LIN {X 0,Y 440.181,Z 736.749,A -85,B 0,C 180,E1 21310.496,E2 21310.496} C_VEL
LIN {X 0,Y 440.061,Z 740.552,A -85,B 0,C 180,E1 21308.405,E2 21308.405} C_VEL
LIN {X 0,Y 440.015,Z 742.533,A -85,B 0,C 180,E1 21306.286,E2 21306.286} C_VEL
LIN {X 0,Y 440.014,Z 742.803,A -85,B 0,C 180,E1 21304.135,E2 21304.135} C_VEL
LIN {X 0,Y 440.046,Z 741.335,A -85,B 0,C 180,E1 21302.093,E2 21302.093} C_VEL
LIN {X 0,Y 440.151,Z 738.009,A -85,B 0,C 180,E1 21299.94,E2 21299.94} C_VEL
LIN {X 0,Y 440.36,Z 733.034,A -85,B 0,C 180,E1 21297.908,E2 21297.908} C_VEL
LIN {X 0,Y 440.738,Z 726.189,A -85,B 0,C 180,E1 21295.899,E2 21295.899} C_VEL
LIN {X 0,Y 441.277,Z 718.01,A -85,B 0,C 180,E1 21294.069,E2 21294.069} C_VEL
LIN {X 0,Y 442.008,Z 707.793,A -85,B 0,C 180,E1 21292.276,E2 21292.276} C_VEL
LIN {X 0,Y 442.843,Z 696.61,A -85,B 0,C 180,E1 21290.715,E2 21290.715} C_VEL
LIN {X 0,Y 443.748,Z 683.902,A -85,B 0,C 180,E1 21289.299,E2 21289.299} C_VEL
LIN {X 0,Y 444.656,Z 670.333,A -85,B 0,C 180,E1 21288.099,E2 21288.099} C_VEL
LIN {X 0,Y 445.545,Z 654.948,A -85,B 0,C 180,E1 21287.053,E2 21287.053} C_VEL
LIN {X 0,Y 446.221,Z 639.636,A -85,B 0,C 180,E1 21286.284,E2 21286.284} C_VEL
LIN {X 0,Y 446.712,Z 622.753,A -85,B 0,C 180,E1 21285.709,E2 21285.709} C_VEL
LIN {X 0,Y 447.044,Z 598.324,A -85,B 0,C 180,E1 21285.256,E2 21285.256} C_VEL
LIN {X 0,Y 448.29,Z 488.008,A -85,B 0,C 180,E1 21283.44,E2 21283.44} C_VEL
LIN {X 0,Y 447.015,Z 476.916,A -85,B 0,C 180,E1 21283.152,E2 21283.152} C_VEL
LIN {X 0,Y 448.557,Z 433.644,A -85,B 0,C 180,E1 21279.442,E2 21279.442} C_VEL
LIN {X 0,Y 450.183,Z 391.513,A -85,B 0,C 180,E1 21275.842,E2 21275.842} C_VEL
LIN {X 0,Y 451.444,Z 352.894,A -85,B 0,C 180,E1 21272.562,E2 21272.562} C_VEL
LIN {X 0,Y 452.462,Z 314.159,A -85,B 0,C 180,E1 21269.27,E2 21269.27} C_VEL
LIN {X 0,Y 446.407,Z 295.705,A -85,B 0,C 180,E1 21267.189,E2 21267.189} C_VEL
LIN {X 0,Y 441.254,Z 281.906,A -85,B 0,C 180,E1 21265.502,E2 21265.502} C_VEL
LIN {X 0,Y 441.178,Z 281.529,A -85,B 0,C 180,E1 21265.076,E2 21265.076} C_VEL
LIN {X 0,Y 441.198,Z 281.522,A -85,B 0,C 180,E1 21261.348,E2 21261.348} C_VEL
LIN {X 0,Y 441.197,Z 281.527,A -85,B 0,C 180,E1 21257.543,E2 21257.543} C_VEL
LIN {X 0,Y 441.185,Z 281.533,A -85,B 0,C 180,E1 21253.767,E2 21253.767} C_VEL
LIN {X 0,Y 441.166,Z 281.531,A -85,B 0,C 180,E1 21250.051,E2 21250.051} C_VEL
LIN {X 0,Y 441.16,Z 281.529,A -85,B 0,C 180,E1 21246.377,E2 21246.377} C_VEL
LIN {X 0,Y 441.167,Z 281.529,A -85,B 0,C 180,E1 21242.598,E2 21242.598} C_VEL
LIN {X 0,Y 441.191,Z 281.524,A -85,B 0,C 180,E1 21238.962,E2 21238.962} C_VEL
LIN {X 0,Y 441.199,Z 281.529,A -85,B 0,C 180,E1 21235.191,E2 21235.191} C_VEL
LIN {X 0,Y 441.196,Z 281.528,A -85,B 0,C 180,E1 21231.398,E2 21231.398} C_VEL
LIN {X 0,Y 441.18,Z 281.528,A -85,B 0,C 180,E1 21227.621,E2 21227.621} C_VEL
LIN {X 0,Y 441.166,Z 281.526,A -85,B 0,C 180,E1 21223.928,E2 21223.928} C_VEL
LIN {X 0,Y 441.164,Z 281.528,A -85,B 0,C 180,E1 21220.126,E2 21220.126} C_VEL
LIN {X 0,Y 441.173,Z 281.528,A -85,B 0,C 180,E1 21216.351,E2 21216.351} C_VEL
LIN {X 0,Y 441.191,Z 281.525,A -85,B 0,C 180,E1 21212.61,E2 21212.61} C_VEL
LIN {X 0,Y 441.201,Z 281.527,A -85,B 0,C 180,E1 21208.889,E2 21208.889} C_VEL
LIN {X 0,Y 441.198,Z 281.531,A -85,B 0,C 180,E1 21205.119,E2 21205.119} C_VEL
LIN {X 0,Y 441.192,Z 281.531,A -85,B 0,C 180,E1 21201.282,E2 21201.282} C_VEL
LIN {X 0,Y 441.177,Z 281.532,A -85,B 0,C 180,E1 21197.518,E2 21197.518} C_VEL
LIN {X 0,Y 441.171,Z 281.531,A -85,B 0,C 180,E1 21193.726,E2 21193.726} C_VEL
LIN {X 0,Y 441.247,Z 281.87,A -85,B 0,C 180,E1 21192.618,E2 21192.618} C_VEL
LIN {X 0,Y 450.274,Z 303.715,A -85,B 0,C 180,E1 21189.499,E2 21189.499} C_VEL
LIN {X 0,Y 455.991,Z 317.99,A -85,B 0,C 180,E1 21187.668,E2 21187.668} C_VEL
LIN {X 0,Y 460.666,Z 327.189,A -85,B 0,C 180,E1 21187.056,E2 21187.056} C_VEL
LIN {X 0,Y 462.807,Z 343.497,A -85,B 0,C 180,E1 21186.538,E2 21186.538} C_VEL
LIN {X 0,Y 457.811,Z 535.941,A -85,B 0,C 180,E1 21183.072,E2 21183.072} C_VEL
LIN {X 0,Y 456.712,Z 578.69,A -85,B 0,C 180,E1 21182.281,E2 21182.281} C_VEL
LIN {X 0,Y 455.661,Z 599.497,A -85,B 0,C 180,E1 21181.679,E2 21181.679} C_VEL
LIN {X 0,Y 454.252,Z 620.653,A -85,B 0,C 180,E1 21180.816,E2 21180.816} C_VEL
LIN {X 0,Y 452.631,Z 640.786,A -85,B 0,C 180,E1 21179.736,E2 21179.736} C_VEL
LIN {X 0,Y 450.918,Z 659.614,A -85,B 0,C 180,E1 21178.471,E2 21178.471} C_VEL
LIN {X 0,Y 449.126,Z 677.545,A -85,B 0,C 180,E1 21177.008,E2 21177.008} C_VEL
LIN {X 0,Y 447.343,Z 694.663,A -85,B 0,C 180,E1 21175.334,E2 21175.334} C_VEL
LIN {X 0,Y 445.58,Z 711.241,A -85,B 0,C 180,E1 21173.398,E2 21173.398} C_VEL
LIN {X 0,Y 444.067,Z 725.727,A -85,B 0,C 180,E1 21171.391,E2 21171.391} C_VEL
LIN {X 0,Y 442.781,Z 738.828,A -85,B 0,C 180,E1 21169.248,E2 21169.248} C_VEL
LIN {X 0,Y 441.743,Z 750.531,A -85,B 0,C 180,E1 21166.975,E2 21166.975} C_VEL
LIN {X 0,Y 440.958,Z 760.738,A -85,B 0,C 180,E1 21164.576,E2 21164.576} C_VEL
LIN {X 0,Y 440.444,Z 769.059,A -85,B 0,C 180,E1 21162.186,E2 21162.186} C_VEL
LIN {X 0,Y 440.125,Z 776.357,A -85,B 0,C 180,E1 21159.544,E2 21159.544} C_VEL
LIN {X 0,Y 439.984,Z 781.551,A -85,B 0,C 180,E1 21157.047,E2 21157.047} C_VEL
LIN {X 0,Y 439.941,Z 785.113,A -85,B 0,C 180,E1 21154.561,E2 21154.561} C_VEL
LIN {X 0,Y 439.94,Z 787.077,A -85,B 0,C 180,E1 21152.082,E2 21152.082} C_VEL
LIN {X 0,Y 439.937,Z 787.552,A -85,B 0,C 180,E1 21149.478,E2 21149.478} C_VEL
LIN {X 0,Y 439.937,Z 786.489,A -85,B 0,C 180,E1 21147.002,E2 21147.002} C_VEL
LIN {X 0,Y 439.952,Z 783.805,A -85,B 0,C 180,E1 21144.513,E2 21144.513} C_VEL
LIN {X 0,Y 440.044,Z 779.312,A -85,B 0,C 180,E1 21141.9,E2 21141.9} C_VEL
LIN {X 0,Y 440.252,Z 772.933,A -85,B 0,C 180,E1 21139.266,E2 21139.266} C_VEL
LIN {X 0,Y 440.634,Z 764.984,A -85,B 0,C 180,E1 21136.75,E2 21136.75} C_VEL
LIN {X 0,Y 441.243,Z 755.554,A -85,B 0,C 180,E1 21134.355,E2 21134.355} C_VEL
LIN {X 0,Y 442.122,Z 743.965,A -85,B 0,C 180,E1 21131.95,E2 21131.95} C_VEL
LIN {X 0,Y 443.172,Z 731.504,A -85,B 0,C 180,E1 21129.805,E2 21129.805} C_VEL
LIN {X 0,Y 444.435,Z 717.672,A -85,B 0,C 180,E1 21127.792,E2 21127.792} C_VEL
LIN {X 0,Y 445.876,Z 702.126,A -85,B 0,C 180,E1 21125.878,E2 21125.878} C_VEL
LIN {X 0,Y 447.474,Z 684.889,A -85,B 0,C 180,E1 21124.097,E2 21124.097} C_VEL
LIN {X 0,Y 449.047,Z 666.984,A -85,B 0,C 180,E1 21122.553,E2 21122.553} C_VEL
LIN {X 0,Y 450.605,Z 648.2,A -85,B 0,C 180,E1 21121.215,E2 21121.215} C_VEL
LIN {X 0,Y 452.045,Z 628.603,A -85,B 0,C 180,E1 21120.08,E2 21120.08} C_VEL
LIN {X 0,Y 453.369,Z 607.681,A -85,B 0,C 180,E1 21119.133,E2 21119.133} C_VEL
LIN {X 0,Y 454.47,Z 585.842,A -85,B 0,C 180,E1 21118.407,E2 21118.407} C_VEL
LIN {X 0,Y 455.219,Z 563.267,A -85,B 0,C 180,E1 21117.912,E2 21117.912} C_VEL
LIN {X 0,Y 457.443,Z 471.715,A -85,B 0,C 180,E1 21116.219,E2 21116.219} C_VEL
LIN {X 0,Y 460.734,Z 385.677,A -85,B 0,C 180,E1 21114.431,E2 21114.431} C_VEL
LIN {X 0,Y 462.815,Z 341.137,A -85,B 0,C 180,E1 21113.409,E2 21113.409} C_VEL
LIN {X 0,Y 461.409,Z 327.079,A -85,B 0,C 180,E1 21112.807,E2 21112.807} C_VEL
LIN {X 0,Y 459.208,Z 322.242,A -85,B 0,C 180,E1 21112.322,E2 21112.322} C_VEL
LIN {X 0,Y 456.915,Z 314.351,A -85,B 0,C 180,E1 21110.932,E2 21110.932} C_VEL
LIN {X 0,Y 454.658,Z 308.19,A -85,B 0,C 180,E1 21109.543,E2 21109.543} C_VEL
LIN {X 0,Y 453.091,Z 304.346,A -85,B 0,C 180,E1 21108.425,E2 21108.425} C_VEL
LIN {X 0,Y 451.999,Z 301.525,A -85,B 0,C 180,E1 21107.397,E2 21107.397} C_VEL
LIN {X 0,Y 450.664,Z 298.499,A -85,B 0,C 180,E1 21105.594,E2 21105.594} C_VEL
LIN {X 0,Y 450.382,Z 297.678,A -85,B 0,C 180,E1 21104.549,E2 21104.549} C_VEL
LIN {X 0,Y 450.505,Z 297.961,A -85,B 0,C 180,E1 21102.91,E2 21102.91} C_VEL
LIN {X 0,Y 451.405,Z 300.859,A -85,B 0,C 180,E1 21100.946,E2 21100.946} C_VEL
LIN {X 0,Y 452.242,Z 302.678,A -85,B 0,C 180,E1 21100.095,E2 21100.095} C_VEL
LIN {X 0,Y 453.759,Z 306.663,A -85,B 0,C 180,E1 21098.735,E2 21098.735} C_VEL
LIN {X 0,Y 455.605,Z 311.582,A -85,B 0,C 180,E1 21097.397,E2 21097.397} C_VEL
LIN {X 0,Y 458.153,Z 319.894,A -85,B 0,C 180,E1 21095.64,E2 21095.64} C_VEL
LIN {X 0,Y 459.651,Z 326.416,A -85,B 0,C 180,E1 21094.509,E2 21094.509} C_VEL
LIN {X 0,Y 458.028,Z 338.193,A -85,B 0,C 180,E1 21093.261,E2 21093.261} C_VEL
LIN {X 0,Y 460.688,Z 358.394,A -85,B 0,C 180,E1 21092.208,E2 21092.208} C_VEL
LIN {X 0,Y 461.626,Z 369.193,A -85,B 0,C 180,E1 21091.757,E2 21091.757} C_VEL
LIN {X 0,Y 456.809,Z 456.691,A -85,B 0,C 180,E1 21089.751,E2 21089.751} C_VEL
LIN {X 0,Y 453.689,Z 542.646,A -85,B 0,C 180,E1 21087.956,E2 21087.956} C_VEL
LIN {X 0,Y 452.772,Z 568.529,A -85,B 0,C 180,E1 21087.378,E2 21087.378} C_VEL
LIN {X 0,Y 451.765,Z 588.323,A -85,B 0,C 180,E1 21086.697,E2 21086.697} C_VEL
LIN {X 0,Y 450.577,Z 606.905,A -85,B 0,C 180,E1 21085.828,E2 21085.828} C_VEL
LIN {X 0,Y 449.224,Z 625.06,A -85,B 0,C 180,E1 21084.736,E2 21084.736} C_VEL
LIN {X 0,Y 447.734,Z 642.969,A -85,B 0,C 180,E1 21083.388,E2 21083.388} C_VEL
LIN {X 0,Y 446.223,Z 659.644,A -85,B 0,C 180,E1 21081.836,E2 21081.836} C_VEL
LIN {X 0,Y 444.779,Z 674.825,A -85,B 0,C 180,E1 21080.117,E2 21080.117} C_VEL
LIN {X 0,Y 443.489,Z 688.388,A -85,B 0,C 180,E1 21078.263,E2 21078.263} C_VEL
LIN {X 0,Y 442.379,Z 700.441,A -85,B 0,C 180,E1 21076.275,E2 21076.275} C_VEL
LIN {X 0,Y 441.483,Z 711.005,A -85,B 0,C 180,E1 21074.158,E2 21074.158} C_VEL
LIN {X 0,Y 440.847,Z 719.619,A -85,B 0,C 180,E1 21072.043,E2 21072.043} C_VEL
LIN {X 0,Y 440.381,Z 727.255,A -85,B 0,C 180,E1 21069.672,E2 21069.672} C_VEL
LIN {X 0,Y 440.121,Z 733.018,A -85,B 0,C 180,E1 21067.309,E2 21067.309} C_VEL
LIN {X 0,Y 439.997,Z 737.235,A -85,B 0,C 180,E1 21064.823,E2 21064.823} C_VEL
LIN {X 0,Y 439.954,Z 739.675,A -85,B 0,C 180,E1 21062.344,E2 21062.344} C_VEL
LIN {X 0,Y 439.951,Z 740.425,A -85,B 0,C 180,E1 21059.869,E2 21059.869} C_VEL
LIN {X 0,Y 439.953,Z 739.489,A -85,B 0,C 180,E1 21057.394,E2 21057.394} C_VEL
LIN {X 0,Y 439.993,Z 736.836,A -85,B 0,C 180,E1 21054.915,E2 21054.915} C_VEL
LIN {X 0,Y 440.118,Z 732.414,A -85,B 0,C 180,E1 21052.428,E2 21052.428} C_VEL
LIN {X 0,Y 440.407,Z 726.08,A -85,B 0,C 180,E1 21049.932,E2 21049.932} C_VEL
LIN {X 0,Y 440.892,Z 718.138,A -85,B 0,C 180,E1 21047.558,E2 21047.558} C_VEL
LIN {X 0,Y 441.611,Z 708.667,A -85,B 0,C 180,E1 21045.31,E2 21045.31} C_VEL
LIN {X 0,Y 442.571,Z 697.708,A -85,B 0,C 180,E1 21043.191,E2 21043.191} C_VEL
LIN {X 0,Y 443.755,Z 685.267,A -85,B 0,C 180,E1 21041.203,E2 21041.203} C_VEL
LIN {X 0,Y 445.136,Z 671.283,A -85,B 0,C 180,E1 21039.35,E2 21039.35} C_VEL
LIN {X 0,Y 446.614,Z 656.284,A -85,B 0,C 180,E1 21037.699,E2 21037.699} C_VEL
LIN {X 0,Y 448.114,Z 640.389,A -85,B 0,C 180,E1 21036.25,E2 21036.25} C_VEL
LIN {X 0,Y 449.573,Z 623.714,A -85,B 0,C 180,E1 21035.003,E2 21035.003} C_VEL
LIN {X 0,Y 450.969,Z 605.565,A -85,B 0,C 180,E1 21033.917,E2 21033.917} C_VEL
LIN {X 0,Y 452.193,Z 586.81,A -85,B 0,C 180,E1 21033.054,E2 21033.054} C_VEL
LIN {X 0,Y 453.148,Z 567.759,A -85,B 0,C 180,E1 21032.418,E2 21032.418} C_VEL
LIN {X 0,Y 453.837,Z 546.607,A -85,B 0,C 180,E1 21031.963,E2 21031.963} C_VEL
LIN {X 0,Y 458.256,Z 366.504,A -85,B 0,C 180,E1 21028.685,E2 21028.685} C_VEL
LIN {X 0,Y 454.172,Z 340.574,A -85,B 0,C 180,E1 21027.787,E2 21027.787} C_VEL
LIN {X 0,Y 455.736,Z 321.368,A -85,B 0,C 180,E1 21025.928,E2 21025.928} C_VEL
LIN {X 0,Y 449.365,Z 303.02,A -85,B 0,C 180,E1 21023.393,E2 21023.393} C_VEL
LIN {X 0,Y 442.233,Z 284.592,A -85,B 0,C 180,E1 21020.647,E2 21020.647} C_VEL
LIN {X 0,Y 441.199,Z 281.714,A -85,B 0,C 180,E1 21020.149,E2 21020.149} C_VEL
LIN {X 0,Y 441.193,Z 281.525,A -85,B 0,C 180,E1 21016.487,E2 21016.487} C_VEL
LIN {X 0,Y 441.195,Z 281.525,A -85,B 0,C 180,E1 21012.658,E2 21012.658} C_VEL
LIN {X 0,Y 441.192,Z 281.529,A -85,B 0,C 180,E1 21009.612,E2 21009.612} C_VEL
LIN {X 0,Y 440.226,Z 281.651,A -85,B 0,C 180,E1 21008.611,E2 21008.611} C_VEL
LIN {X 0,Y 433.688,Z 282.466,A -85,B 0,C 180,E1 21005.722,E2 21005.722} C_VEL
LIN {X 0,Y 433.246,Z 282.517,A -85,B 0,C 180,E1 21005.059,E2 21005.059} C_VEL
LIN {X 0,Y 433.246,Z 282.516,A -85,B 0,C 180,E1 21001.284,E2 21001.284} C_VEL
LIN {X 0,Y 433.248,Z 282.519,A -85,B 0,C 180,E1 20997.489,E2 20997.489} C_VEL
LIN {X 0,Y 433.251,Z 282.513,A -85,B 0,C 180,E1 20993.677,E2 20993.677} C_VEL
LIN {X 0,Y 433.259,Z 282.516,A -85,B 0,C 180,E1 20989.973,E2 20989.973} C_VEL
LIN {X 0,Y 433.254,Z 282.505,A -85,B 0,C 180,E1 20986.079,E2 20986.079} C_VEL
LIN {X 0,Y 433.248,Z 282.789,A -85,B 0,C 180,E1 20985.34,E2 20985.34} C_VEL
LIN {X 0,Y 440.653,Z 303.028,A -85,B 0,C 180,E1 20982.783,E2 20982.783} C_VEL
LIN {X 0,Y 445.747,Z 318.928,A -85,B 0,C 180,E1 20980.927,E2 20980.927} C_VEL
LIN {X 0,Y 444.169,Z 360.129,A -85,B 0,C 180,E1 20977.308,E2 20977.308} C_VEL
LIN {X 0,Y 442.449,Z 402.117,A -85,B 0,C 180,E1 20973.629,E2 20973.629} C_VEL
LIN {X 0,Y 440.609,Z 445.061,A -85,B 0,C 180,E1 20969.871,E2 20969.871} C_VEL
LIN {X 0,Y 439.376,Z 477.348,A -85,B 0,C 180,E1 20967.073,E2 20967.073} C_VEL
LIN {X 0,Y 440.893,Z 492.134,A -85,B 0,C 180,E1 20966.733,E2 20966.733} C_VEL
LIN {X 0,Y 439.134,Z 620.462,A -85,B 0,C 180,E1 20964.571,E2 20964.571} C_VEL
LIN {X 0,Y 438.677,Z 636.459,A -85,B 0,C 180,E1 20964.061,E2 20964.061} C_VEL
LIN {X 0,Y 437.958,Z 652.869,A -85,B 0,C 180,E1 20963.274,E2 20963.274} C_VEL
LIN {X 0,Y 437.106,Z 667.453,A -85,B 0,C 180,E1 20962.311,E2 20962.311} C_VEL
LIN {X 0,Y 436.156,Z 681.295,A -85,B 0,C 180,E1 20961.133,E2 20961.133} C_VEL
LIN {X 0,Y 435.218,Z 693.946,A -85,B 0,C 180,E1 20959.772,E2 20959.772} C_VEL
LIN {X 0,Y 434.264,Z 706.231,A -85,B 0,C 180,E1 20958.109,E2 20958.109} C_VEL
LIN {X 0,Y 433.495,Z 716.267,A -85,B 0,C 180,E1 20956.395,E2 20956.395} C_VEL
LIN {X 0,Y 432.856,Z 725.39,A -85,B 0,C 180,E1 20954.417,E2 20954.417} C_VEL
LIN {X 0,Y 432.451,Z 732.108,A -85,B 0,C 180,E1 20952.51,E2 20952.51} C_VEL
LIN {X 0,Y 432.186,Z 737.739,A -85,B 0,C 180,E1 20950.323,E2 20950.323} C_VEL
LIN {X 0,Y 432.068,Z 741.172,A -85,B 0,C 180,E1 20948.27,E2 20948.27} C_VEL
LIN {X 0,Y 432.025,Z 743.034,A -85,B 0,C 180,E1 20946.09,E2 20946.09} C_VEL
LIN {X 0,Y 432.025,Z 743.18,A -85,B 0,C 180,E1 20944.063,E2 20944.063} C_VEL
LIN {X 0,Y 432.067,Z 741.49,A -85,B 0,C 180,E1 20941.832,E2 20941.832} C_VEL
LIN {X 0,Y 432.191,Z 738.024,A -85,B 0,C 180,E1 20939.648,E2 20939.648} C_VEL
LIN {X 0,Y 432.442,Z 732.785,A -85,B 0,C 180,E1 20937.558,E2 20937.558} C_VEL
LIN {X 0,Y 432.872,Z 725.848,A -85,B 0,C 180,E1 20935.537,E2 20935.537} C_VEL
LIN {X 0,Y 433.495,Z 717.09,A -85,B 0,C 180,E1 20933.608,E2 20933.608} C_VEL
LIN {X 0,Y 434.261,Z 707.32,A -85,B 0,C 180,E1 20931.901,E2 20931.901} C_VEL
LIN {X 0,Y 435.168,Z 695.801,A -85,B 0,C 180,E1 20930.304,E2 20930.304} C_VEL
LIN {X 0,Y 436.161,Z 682.809,A -85,B 0,C 180,E1 20928.861,E2 20928.861} C_VEL
LIN {X 0,Y 437.14,Z 668.595,A -85,B 0,C 180,E1 20927.629,E2 20927.629} C_VEL
LIN {X 0,Y 438.03,Z 653.898,A -85,B 0,C 180,E1 20926.643,E2 20926.643} C_VEL
LIN {X 0,Y 438.742,Z 637.746,A -85,B 0,C 180,E1 20925.855,E2 20925.855} C_VEL
LIN {X 0,Y 439.21,Z 621.585,A -85,B 0,C 180,E1 20925.324,E2 20925.324} C_VEL
LIN {X 0,Y 439.971,Z 565.077,A -85,B 0,C 180,E1 20924.345,E2 20924.345} C_VEL
LIN {X 0,Y 440.868,Z 488.855,A -85,B 0,C 180,E1 20923.064,E2 20923.064} C_VEL
LIN {X 0,Y 439.554,Z 477.444,A -85,B 0,C 180,E1 20922.766,E2 20922.766} C_VEL
LIN {X 0,Y 441.159,Z 434.521,A -85,B 0,C 180,E1 20919.056,E2 20919.056} C_VEL
LIN {X 0,Y 443.037,Z 389.151,A -85,B 0,C 180,E1 20915.135,E2 20915.135} C_VEL
LIN {X 0,Y 444.504,Z 345.174,A -85,B 0,C 180,E1 20911.382,E2 20911.382} C_VEL
LIN {X 0,Y 445.246,Z 316.819,A -85,B 0,C 180,E1 20908.943,E2 20908.943} C_VEL
LIN {X 0,Y 438.945,Z 297.654,A -85,B 0,C 180,E1 20906.737,E2 20906.737} C_VEL
LIN {X 0,Y 433.278,Z 282.866,A -85,B 0,C 180,E1 20904.875,E2 20904.875} C_VEL
LIN {X 0,Y 433.223,Z 282.522,A -85,B 0,C 180,E1 20904.257,E2 20904.257} C_VEL
LIN {X 0,Y 433.219,Z 282.519,A -85,B 0,C 180,E1 20900.446,E2 20900.446} C_VEL
LIN {X 0,Y 433.221,Z 282.523,A -85,B 0,C 180,E1 20896.63,E2 20896.63} C_VEL
LIN {X 0,Y 433.239,Z 282.518,A -85,B 0,C 180,E1 20892.937,E2 20892.937} C_VEL
LIN {X 0,Y 433.257,Z 282.516,A -85,B 0,C 180,E1 20889.163,E2 20889.163} C_VEL
LIN {X 0,Y 433.258,Z 282.52,A -85,B 0,C 180,E1 20885.43,E2 20885.43} C_VEL
LIN {X 0,Y 433.25,Z 282.516,A -85,B 0,C 180,E1 20881.587,E2 20881.587} C_VEL
LIN {X 0,Y 433.231,Z 282.518,A -85,B 0,C 180,E1 20877.884,E2 20877.884} C_VEL
LIN {X 0,Y 433.223,Z 282.52,A -85,B 0,C 180,E1 20874.092,E2 20874.092} C_VEL
LIN {X 0,Y 433.225,Z 282.514,A -85,B 0,C 180,E1 20870.215,E2 20870.215} C_VEL
LIN {X 0,Y 433.229,Z 282.517,A -85,B 0,C 180,E1 20866.385,E2 20866.385} C_VEL
LIN {X 0,Y 433.247,Z 282.516,A -85,B 0,C 180,E1 20862.68,E2 20862.68} C_VEL
LIN {X 0,Y 433.262,Z 282.513,A -85,B 0,C 180,E1 20858.9,E2 20858.9} C_VEL
LIN {X 0,Y 433.261,Z 282.515,A -85,B 0,C 180,E1 20855.082,E2 20855.082} C_VEL
LIN {X 0,Y 433.263,Z 282.518,A -85,B 0,C 180,E1 20851.271,E2 20851.271} C_VEL
LIN {X 0,Y 433.242,Z 282.518,A -85,B 0,C 180,E1 20847.471,E2 20847.471} C_VEL
LIN {X 0,Y 433.229,Z 282.518,A -85,B 0,C 180,E1 20843.785,E2 20843.785} C_VEL
LIN {X 0,Y 433.231,Z 282.518,A -85,B 0,C 180,E1 20839.917,E2 20839.917} C_VEL
LIN {X 0,Y 433.24,Z 282.521,A -85,B 0,C 180,E1 20836.183,E2 20836.183} C_VEL
LIN {X 0,Y 433.28,Z 282.785,A -85,B 0,C 180,E1 20833.395,E2 20833.395} C_VEL
LIN {X 0,Y 442.336,Z 304.575,A -85,B 0,C 180,E1 20830.181,E2 20830.181} C_VEL
LIN {X 0,Y 447.798,Z 318.027,A -85,B 0,C 180,E1 20828.398,E2 20828.398} C_VEL
LIN {X 0,Y 454.373,Z 330.66,A -85,B 0,C 180,E1 20827.533,E2 20827.533} C_VEL
LIN {X 0,Y 456.144,Z 344.815,A -85,B 0,C 180,E1 20827.076,E2 20827.076} C_VEL
LIN {X 0,Y 450.988,Z 527.844,A -85,B 0,C 180,E1 20823.703,E2 20823.703} C_VEL
LIN {X 0,Y 449.614,Z 578.4,A -85,B 0,C 180,E1 20822.755,E2 20822.755} C_VEL
LIN {X 0,Y 448.508,Z 599.317,A -85,B 0,C 180,E1 20822.141,E2 20822.141} C_VEL
LIN {X 0,Y 447.058,Z 619.962,A -85,B 0,C 180,E1 20821.29,E2 20821.29} C_VEL
LIN {X 0,Y 445.444,Z 639.254,A -85,B 0,C 180,E1 20820.25,E2 20820.25} C_VEL
LIN {X 0,Y 443.639,Z 658.179,A -85,B 0,C 180,E1 20818.982,E2 20818.982} C_VEL
LIN {X 0,Y 441.751,Z 676.334,A -85,B 0,C 180,E1 20817.497,E2 20817.497} C_VEL
LIN {X 0,Y 439.792,Z 694.198,A -85,B 0,C 180,E1 20815.735,E2 20815.735} C_VEL
LIN {X 0,Y 437.917,Z 710.869,A -85,B 0,C 180,E1 20813.763,E2 20813.763} C_VEL
LIN {X 0,Y 436.365,Z 724.971,A -85,B 0,C 180,E1 20811.788,E2 20811.788} C_VEL
LIN {X 0,Y 434.99,Z 738.152,A -85,B 0,C 180,E1 20809.607,E2 20809.607} C_VEL
LIN {X 0,Y 433.82,Z 750.534,A -85,B 0,C 180,E1 20807.156,E2 20807.156} C_VEL
LIN {X 0,Y 432.96,Z 761.231,A -85,B 0,C 180,E1 20804.578,E2 20804.578} C_VEL
LIN {X 0,Y 432.416,Z 769.799,A -85,B 0,C 180,E1 20802.01,E2 20802.01} C_VEL
LIN {X 0,Y 432.115,Z 776.509,A -85,B 0,C 180,E1 20799.454,E2 20799.454} C_VEL
LIN {X 0,Y 431.987,Z 781.745,A -85,B 0,C 180,E1 20796.778,E2 20796.778} C_VEL
LIN {X 0,Y 431.948,Z 785.092,A -85,B 0,C 180,E1 20794.246,E2 20794.246} C_VEL
LIN {X 0,Y 431.946,Z 786.854,A -85,B 0,C 180,E1 20791.723,E2 20791.723} C_VEL
LIN {X 0,Y 431.953,Z 787.069,A -85,B 0,C 180,E1 20789.203,E2 20789.203} C_VEL
LIN {X 0,Y 431.945,Z 785.687,A -85,B 0,C 180,E1 20786.548,E2 20786.548} C_VEL
LIN {X 0,Y 431.975,Z 782.803,A -85,B 0,C 180,E1 20784.02,E2 20784.02} C_VEL
LIN {X 0,Y 432.075,Z 777.952,A -85,B 0,C 180,E1 20781.348,E2 20781.348} C_VEL
LIN {X 0,Y 432.298,Z 771.561,A -85,B 0,C 180,E1 20778.796,E2 20778.796} C_VEL
LIN {X 0,Y 432.741,Z 763.295,A -85,B 0,C 180,E1 20776.231,E2 20776.231} C_VEL
LIN {X 0,Y 433.418,Z 753.53,A -85,B 0,C 180,E1 20773.79,E2 20773.79} C_VEL
LIN {X 0,Y 434.338,Z 742.313,A -85,B 0,C 180,E1 20771.476,E2 20771.476} C_VEL
LIN {X 0,Y 435.481,Z 729.664,A -85,B 0,C 180,E1 20769.292,E2 20769.292} C_VEL
LIN {X 0,Y 436.89,Z 715.019,A -85,B 0,C 180,E1 20767.174,E2 20767.174} C_VEL
LIN {X 0,Y 438.368,Z 699.902,A -85,B 0,C 180,E1 20765.328,E2 20765.328} C_VEL
LIN {X 0,Y 439.988,Z 683.393,A -85,B 0,C 180,E1 20763.622,E2 20763.622} C_VEL
LIN {X 0,Y 441.659,Z 665.268,A -85,B 0,C 180,E1 20762.054,E2 20762.054} C_VEL
LIN {X 0,Y 443.315,Z 646.208,A -85,B 0,C 180,E1 20760.696,E2 20760.696} C_VEL
LIN {X 0,Y 444.827,Z 626.726,A -85,B 0,C 180,E1 20759.57,E2 20759.57} C_VEL
LIN {X 0,Y 446.189,Z 606.313,A -85,B 0,C 180,E1 20758.645,E2 20758.645} C_VEL
LIN {X 0,Y 447.344,Z 585.056,A -85,B 0,C 180,E1 20757.932,E2 20757.932} C_VEL
LIN {X 0,Y 448.156,Z 562.417,A -85,B 0,C 180,E1 20757.423,E2 20757.423} C_VEL
LIN {X 0,Y 450.521,Z 476.99,A -85,B 0,C 180,E1 20755.78,E2 20755.78} C_VEL
LIN {X 0,Y 454.064,Z 394.65,A -85,B 0,C 180,E1 20753.998,E2 20753.998} C_VEL
LIN {X 0,Y 456.926,Z 342.616,A -85,B 0,C 180,E1 20752.753,E2 20752.753} C_VEL
LIN {X 0,Y 455.948,Z 331.016,A -85,B 0,C 180,E1 20752.236,E2 20752.236} C_VEL
LIN {X 0,Y 452.344,Z 323.393,A -85,B 0,C 180,E1 20751.396,E2 20751.396} C_VEL
LIN {X 0,Y 450.124,Z 316.137,A -85,B 0,C 180,E1 20749.895,E2 20749.895} C_VEL
LIN {X 0,Y 448.031,Z 310.491,A -85,B 0,C 180,E1 20748.314,E2 20748.314} C_VEL
LIN {X 0,Y 446.844,Z 307.472,A -85,B 0,C 180,E1 20747.137,E2 20747.137} C_VEL
LIN {X 0,Y 445.826,Z 304.501,A -85,B 0,C 180,E1 20745.233,E2 20745.233} C_VEL
LIN {X 0,Y 445.598,Z 304.07,A -85,B 0,C 180,E1 20743.54,E2 20743.54} C_VEL
LIN {X 0,Y 445.761,Z 305.238,A -85,B 0,C 180,E1 20742.25,E2 20742.25} C_VEL
LIN {X 0,Y 446.996,Z 308.181,A -85,B 0,C 180,E1 20740.442,E2 20740.442} C_VEL
LIN {X 0,Y 448.407,Z 312.469,A -85,B 0,C 180,E1 20738.903,E2 20738.903} C_VEL
LIN {X 0,Y 450.359,Z 318.322,A -85,B 0,C 180,E1 20737.307,E2 20737.307} C_VEL
LIN {X 0,Y 452.74,Z 326.881,A -85,B 0,C 180,E1 20735.508,E2 20735.508} C_VEL
LIN {X 0,Y 453.286,Z 330.32,A -85,B 0,C 180,E1 20734.918,E2 20734.918} C_VEL
LIN {X 0,Y 452.239,Z 337.786,A -85,B 0,C 180,E1 20734.121,E2 20734.121} C_VEL
LIN {X 0,Y 454.73,Z 358.347,A -85,B 0,C 180,E1 20732.959,E2 20732.959} C_VEL
LIN {X 0,Y 455.701,Z 370.503,A -85,B 0,C 180,E1 20732.414,E2 20732.414} C_VEL
LIN {X 0,Y 450.401,Z 454.66,A -85,B 0,C 180,E1 20730.388,E2 20730.388} C_VEL
LIN {X 0,Y 446.946,Z 535.528,A -85,B 0,C 180,E1 20728.603,E2 20728.603} C_VEL
LIN {X 0,Y 445.747,Z 567.218,A -85,B 0,C 180,E1 20727.891,E2 20727.891} C_VEL
LIN {X 0,Y 444.656,Z 587.344,A -85,B 0,C 180,E1 20727.199,E2 20727.199} C_VEL
LIN {X 0,Y 443.348,Z 606.589,A -85,B 0,C 180,E1 20726.292,E2 20726.292} C_VEL
LIN {X 0,Y 441.885,Z 625.098,A -85,B 0,C 180,E1 20725.164,E2 20725.164} C_VEL
LIN {X 0,Y 440.346,Z 642.497,A -85,B 0,C 180,E1 20723.839,E2 20723.839} C_VEL
LIN {X 0,Y 438.777,Z 658.936,A -85,B 0,C 180,E1 20722.304,E2 20722.304} C_VEL
LIN {X 0,Y 437.236,Z 674.245,A -85,B 0,C 180,E1 20720.568,E2 20720.568} C_VEL
LIN {X 0,Y 435.822,Z 688.217,A -85,B 0,C 180,E1 20718.646,E2 20718.646} C_VEL
LIN {X 0,Y 434.601,Z 700.641,A -85,B 0,C 180,E1 20716.575,E2 20716.575} C_VEL
LIN {X 0,Y 433.639,Z 711.27,A -85,B 0,C 180,E1 20714.419,E2 20714.419} C_VEL
LIN {X 0,Y 432.914,Z 720.399,A -85,B 0,C 180,E1 20712.132,E2 20712.132} C_VEL
LIN {X 0,Y 432.446,Z 727.626,A -85,B 0,C 180,E1 20709.851,E2 20709.851} C_VEL
LIN {X 0,Y 432.157,Z 733.425,A -85,B 0,C 180,E1 20707.444,E2 20707.444} C_VEL
LIN {X 0,Y 432.019,Z 737.66,A -85,B 0,C 180,E1 20704.912,E2 20704.912} C_VEL
LIN {X 0,Y 431.968,Z 740.113,A -85,B 0,C 180,E1 20702.387,E2 20702.387} C_VEL
LIN {X 0,Y 431.962,Z 740.853,A -85,B 0,C 180,E1 20699.867,E2 20699.867} C_VEL
LIN {X 0,Y 431.965,Z 739.896,A -85,B 0,C 180,E1 20697.346,E2 20697.346} C_VEL
LIN {X 0,Y 432.011,Z 737.223,A -85,B 0,C 180,E1 20694.821,E2 20694.821} C_VEL
LIN {X 0,Y 432.149,Z 732.756,A -85,B 0,C 180,E1 20692.287,E2 20692.287} C_VEL
LIN {X 0,Y 432.446,Z 726.765,A -85,B 0,C 180,E1 20689.879,E2 20689.879} C_VEL
LIN {X 0,Y 432.96,Z 718.88,A -85,B 0,C 180,E1 20687.462,E2 20687.462} C_VEL
LIN {X 0,Y 433.719,Z 709.466,A -85,B 0,C 180,E1 20685.173,E2 20685.173} C_VEL
LIN {X 0,Y 434.73,Z 698.574,A -85,B 0,C 180,E1 20683.016,E2 20683.016} C_VEL
LIN {X 0,Y 435.975,Z 686.215,A -85,B 0,C 180,E1 20680.994,E2 20680.994} C_VEL
LIN {X 0,Y 437.425,Z 672.336,A -85,B 0,C 180,E1 20679.109,E2 20679.109} C_VEL
LIN {X 0,Y 438.965,Z 657.587,A -85,B 0,C 180,E1 20677.442,E2 20677.442} C_VEL
LIN {X 0,Y 440.547,Z 641.772,A -85,B 0,C 180,E1 20675.958,E2 20675.958} C_VEL
LIN {X 0,Y 442.133,Z 624.598,A -85,B 0,C 180,E1 20674.642,E2 20674.642} C_VEL
LIN {X 0,Y 443.568,Z 607.09,A -85,B 0,C 180,E1 20673.564,E2 20673.564} C_VEL
LIN {X 0,Y 444.898,Z 587.883,A -85,B 0,C 180,E1 20672.652,E2 20672.652} C_VEL
LIN {X 0,Y 445.932,Z 568.563,A -85,B 0,C 180,E1 20671.987,E2 20671.987} C_VEL
LIN {X 0,Y 446.686,Z 547.242,A -85,B 0,C 180,E1 20671.513,E2 20671.513} C_VEL
LIN {X 0,Y 451.439,Z 367.771,A -85,B 0,C 180,E1 20668.173,E2 20668.173} C_VEL
LIN {X 0,Y 447.208,Z 340.629,A -85,B 0,C 180,E1 20667.21,E2 20667.21} C_VEL
LIN {X 0,Y 448.49,Z 324.02,A -85,B 0,C 180,E1 20665.577,E2 20665.577} C_VEL
LIN {X 0,Y 442.075,Z 305.546,A -85,B 0,C 180,E1 20662.978,E2 20662.978} C_VEL
LIN {X 0,Y 434.556,Z 286.085,A -85,B 0,C 180,E1 20660.014,E2 20660.014} C_VEL
LIN {X 0,Y 433.271,Z 282.713,A -85,B 0,C 180,E1 20659.422,E2 20659.422} C_VEL
LIN {X 0,Y 433.242,Z 282.512,A -85,B 0,C 180,E1 20655.63,E2 20655.63} C_VEL
LIN {X 0,Y 433.246,Z 282.52,A -85,B 0,C 180,E1 20651.803,E2 20651.803} C_VEL
LIN {X 0,Y 433.25,Z 282.517,A -85,B 0,C 180,E1 20648.039,E2 20648.039} C_VEL
LIN {X 0,Y 433.246,Z 282.517,A -85,B 0,C 180,E1 20645.059,E2 20645.059} C_VEL
LIN {X 0,Y 432.246,Z 282.642,A -85,B 0,C 180,E1 20644.04,E2 20644.04} C_VEL
LIN {X 0,Y 425.723,Z 283.455,A -85,B 0,C 180,E1 20641.097,E2 20641.097} C_VEL
LIN {X 0,Y 425.317,Z 283.497,A -85,B 0,C 180,E1 20640.422,E2 20640.422} C_VEL
LIN {X 0,Y 425.297,Z 283.507,A -85,B 0,C 180,E1 20636.683,E2 20636.683} C_VEL
LIN {X 0,Y 425.287,Z 283.51,A -85,B 0,C 180,E1 20632.837,E2 20632.837} C_VEL
LIN {X 0,Y 425.278,Z 283.509,A -85,B 0,C 180,E1 20629.066,E2 20629.066} C_VEL
LIN {X 0,Y 425.351,Z 283.75,A -85,B 0,C 180,E1 20625.964,E2 20625.964} C_VEL
LIN {X 0,Y 432.833,Z 303.892,A -85,B 0,C 180,E1 20623.357,E2 20623.357} C_VEL
LIN {X 0,Y 438.539,Z 321.631,A -85,B 0,C 180,E1 20621.242,E2 20621.242} C_VEL
LIN {X 0,Y 436.845,Z 363.163,A -85,B 0,C 180,E1 20617.564,E2 20617.564} C_VEL
LIN {X 0,Y 435.001,Z 404.586,A -85,B 0,C 180,E1 20613.889,E2 20613.889} C_VEL
LIN {X 0,Y 433.138,Z 446.443,A -85,B 0,C 180,E1 20610.2,E2 20610.2} C_VEL
LIN {X 0,Y 431.886,Z 477.718,A -85,B 0,C 180,E1 20607.467,E2 20607.467} C_VEL
LIN {X 0,Y 433.448,Z 492.914,A -85,B 0,C 180,E1 20607.109,E2 20607.109} C_VEL
LIN {X 0,Y 431.587,Z 620.801,A -85,B 0,C 180,E1 20604.918,E2 20604.918} C_VEL
LIN {X 0,Y 431.105,Z 636.833,A -85,B 0,C 180,E1 20604.398,E2 20604.398} C_VEL
LIN {X 0,Y 430.349,Z 653.229,A -85,B 0,C 180,E1 20603.599,E2 20603.599} C_VEL
LIN {X 0,Y 429.475,Z 667.498,A -85,B 0,C 180,E1 20602.645,E2 20602.645} C_VEL
LIN {X 0,Y 428.443,Z 681.77,A -85,B 0,C 180,E1 20601.412,E2 20601.412} C_VEL
LIN {X 0,Y 427.433,Z 694.579,A -85,B 0,C 180,E1 20600.005,E2 20600.005} C_VEL
LIN {X 0,Y 426.454,Z 706.448,A -85,B 0,C 180,E1 20598.369,E2 20598.369} C_VEL
LIN {X 0,Y 425.661,Z 716.181,A -85,B 0,C 180,E1 20596.693,E2 20596.693} C_VEL
LIN {X 0,Y 424.974,Z 725.234,A -85,B 0,C 180,E1 20594.718,E2 20594.718} C_VEL
LIN {X 0,Y 424.517,Z 732.222,A -85,B 0,C 180,E1 20592.738,E2 20592.738} C_VEL
LIN {X 0,Y 424.22,Z 737.892,A -85,B 0,C 180,E1 20590.525,E2 20590.525} C_VEL
LIN {X 0,Y 424.087,Z 741.451,A -85,B 0,C 180,E1 20588.422,E2 20588.422} C_VEL
LIN {X 0,Y 424.035,Z 743.381,A -85,B 0,C 180,E1 20586.192,E2 20586.192} C_VEL
LIN {X 0,Y 424.036,Z 743.55,A -85,B 0,C 180,E1 20583.989,E2 20583.989} C_VEL
LIN {X 0,Y 424.084,Z 741.82,A -85,B 0,C 180,E1 20581.715,E2 20581.715} C_VEL
LIN {X 0,Y 424.218,Z 738.441,A -85,B 0,C 180,E1 20579.555,E2 20579.555} C_VEL
LIN {X 0,Y 424.504,Z 733.024,A -85,B 0,C 180,E1 20577.361,E2 20577.361} C_VEL
LIN {X 0,Y 424.978,Z 726.004,A -85,B 0,C 180,E1 20575.297,E2 20575.297} C_VEL
LIN {X 0,Y 425.641,Z 717.38,A -85,B 0,C 180,E1 20573.371,E2 20573.371} C_VEL
LIN {X 0,Y 426.485,Z 707.323,A -85,B 0,C 180,E1 20571.594,E2 20571.594} C_VEL
LIN {X 0,Y 427.46,Z 695.706,A -85,B 0,C 180,E1 20569.968,E2 20569.968} C_VEL
LIN {X 0,Y 428.436,Z 683.67,A -85,B 0,C 180,E1 20568.61,E2 20568.61} C_VEL
LIN {X 0,Y 429.46,Z 669.725,A -85,B 0,C 180,E1 20567.368,E2 20567.368} C_VEL
LIN {X 0,Y 430.431,Z 654.607,A -85,B 0,C 180,E1 20566.326,E2 20566.326} C_VEL
LIN {X 0,Y 431.18,Z 638.651,A -85,B 0,C 180,E1 20565.528,E2 20565.528} C_VEL
LIN {X 0,Y 431.689,Z 622.404,A -85,B 0,C 180,E1 20564.977,E2 20564.977} C_VEL
LIN {X 0,Y 432.325,Z 578.125,A -85,B 0,C 180,E1 20564.184,E2 20564.184} C_VEL
LIN {X 0,Y 433.48,Z 489.716,A -85,B 0,C 180,E1 20562.671,E2 20562.671} C_VEL
LIN {X 0,Y 432.105,Z 477.371,A -85,B 0,C 180,E1 20562.327,E2 20562.327} C_VEL
LIN {X 0,Y 433.819,Z 434.461,A -85,B 0,C 180,E1 20558.577,E2 20558.577} C_VEL
LIN {X 0,Y 435.72,Z 390.732,A -85,B 0,C 180,E1 20554.767,E2 20554.767} C_VEL
LIN {X 0,Y 437.267,Z 348.437,A -85,B 0,C 180,E1 20551.117,E2 20551.117} C_VEL
LIN {X 0,Y 438.139,Z 319.782,A -85,B 0,C 180,E1 20548.636,E2 20548.636} C_VEL
LIN {X 0,Y 432.043,Z 301.18,A -85,B 0,C 180,E1 20546.456,E2 20546.456} C_VEL
LIN {X 0,Y 426.068,Z 286.111,A -85,B 0,C 180,E1 20544.543,E2 20544.543} C_VEL
LIN {X 0,Y 425.333,Z 283.825,A -85,B 0,C 180,E1 20544.208,E2 20544.208} C_VEL
LIN {X 0,Y 425.305,Z 283.504,A -85,B 0,C 180,E1 20543.117,E2 20543.117} C_VEL
LIN {X 0,Y 425.319,Z 283.502,A -85,B 0,C 180,E1 20539.359,E2 20539.359} C_VEL
LIN {X 0,Y 425.322,Z 283.497,A -85,B 0,C 180,E1 20535.464,E2 20535.464} C_VEL
LIN {X 0,Y 425.31,Z 283.513,A -85,B 0,C 180,E1 20531.665,E2 20531.665} C_VEL
LIN {X 0,Y 425.299,Z 283.508,A -85,B 0,C 180,E1 20527.838,E2 20527.838} C_VEL
LIN {X 0,Y 425.288,Z 283.507,A -85,B 0,C 180,E1 20524.045,E2 20524.045} C_VEL
LIN {X 0,Y 425.284,Z 283.508,A -85,B 0,C 180,E1 20520.27,E2 20520.27} C_VEL
LIN {X 0,Y 425.288,Z 283.505,A -85,B 0,C 180,E1 20516.496,E2 20516.496} C_VEL
LIN {X 0,Y 425.304,Z 283.504,A -85,B 0,C 180,E1 20512.707,E2 20512.707} C_VEL
LIN {X 0,Y 425.314,Z 283.505,A -85,B 0,C 180,E1 20508.886,E2 20508.886} C_VEL
LIN {X 0,Y 425.325,Z 283.501,A -85,B 0,C 180,E1 20505.014,E2 20505.014} C_VEL
LIN {X 0,Y 425.322,Z 283.501,A -85,B 0,C 180,E1 20501.07,E2 20501.07} C_VEL
LIN {X 0,Y 425.327,Z 283.505,A -85,B 0,C 180,E1 20497.143,E2 20497.143} C_VEL
LIN {X 0,Y 425.314,Z 283.506,A -85,B 0,C 180,E1 20493.29,E2 20493.29} C_VEL
LIN {X 0,Y 425.305,Z 283.507,A -85,B 0,C 180,E1 20489.483,E2 20489.483} C_VEL
LIN {X 0,Y 425.296,Z 283.506,A -85,B 0,C 180,E1 20485.651,E2 20485.651} C_VEL
LIN {X 0,Y 425.293,Z 283.506,A -85,B 0,C 180,E1 20481.808,E2 20481.808} C_VEL
LIN {X 0,Y 425.293,Z 283.51,A -85,B 0,C 180,E1 20477.931,E2 20477.931} C_VEL
LIN {X 0,Y 425.336,Z 283.755,A -85,B 0,C 180,E1 20474.184,E2 20474.184} C_VEL
LIN {X 0,Y 427.659,Z 289.654,A -85,B 0,C 180,E1 20473.235,E2 20473.235} C_VEL
LIN {X 0,Y 435.832,Z 308.948,A -85,B 0,C 180,E1 20470.39,E2 20470.39} C_VEL
LIN {X 0,Y 439.693,Z 318.355,A -85,B 0,C 180,E1 20469.131,E2 20469.131} C_VEL
LIN {X 0,Y 448.026,Z 334.101,A -85,B 0,C 180,E1 20468.008,E2 20468.008} C_VEL
LIN {X 0,Y 449.459,Z 346.034,A -85,B 0,C 180,E1 20467.619,E2 20467.619} C_VEL
LIN {X 0,Y 443.856,Z 532.639,A -85,B 0,C 180,E1 20464.112,E2 20464.112} C_VEL
LIN {X 0,Y 442.508,Z 578.548,A -85,B 0,C 180,E1 20463.228,E2 20463.228} C_VEL
LIN {X 0,Y 441.346,Z 599.416,A -85,B 0,C 180,E1 20462.603,E2 20462.603} C_VEL
LIN {X 0,Y 439.789,Z 620.497,A -85,B 0,C 180,E1 20461.716,E2 20461.716} C_VEL
LIN {X 0,Y 438.006,Z 640.714,A -85,B 0,C 180,E1 20460.599,E2 20460.599} C_VEL
LIN {X 0,Y 436.027,Z 660.308,A -85,B 0,C 180,E1 20459.236,E2 20459.236} C_VEL
LIN {X 0,Y 433.998,Z 678.619,A -85,B 0,C 180,E1 20457.677,E2 20457.677} C_VEL
LIN {X 0,Y 432.12,Z 694.842,A -85,B 0,C 180,E1 20456.022,E2 20456.022} C_VEL
LIN {X 0,Y 430.269,Z 710.469,A -85,B 0,C 180,E1 20454.139,E2 20454.139} C_VEL
LIN {X 0,Y 428.577,Z 725.034,A -85,B 0,C 180,E1 20452.06,E2 20452.06} C_VEL
LIN {X 0,Y 427.131,Z 738.179,A -85,B 0,C 180,E1 20449.84,E2 20449.84} C_VEL
LIN {X 0,Y 425.96,Z 749.911,A -85,B 0,C 180,E1 20447.483,E2 20447.483} C_VEL
LIN {X 0,Y 425.078,Z 760.127,A -85,B 0,C 180,E1 20444.994,E2 20444.994} C_VEL
LIN {X 0,Y 424.495,Z 768.441,A -85,B 0,C 180,E1 20442.513,E2 20442.513} C_VEL
LIN {X 0,Y 424.151,Z 775.609,A -85,B 0,C 180,E1 20439.818,E2 20439.818} C_VEL
LIN {X 0,Y 423.991,Z 780.871,A -85,B 0,C 180,E1 20437.178,E2 20437.178} C_VEL
LIN {X 0,Y 423.954,Z 784.407,A -85,B 0,C 180,E1 20434.598,E2 20434.598} C_VEL
LIN {X 0,Y 423.96,Z 786.292,A -85,B 0,C 180,E1 20432.026,E2 20432.026} C_VEL
LIN {X 0,Y 423.962,Z 786.661,A -85,B 0,C 180,E1 20429.323,E2 20429.323} C_VEL
LIN {X 0,Y 423.954,Z 785.468,A -85,B 0,C 180,E1 20426.754,E2 20426.754} C_VEL
LIN {X 0,Y 423.979,Z 782.673,A -85,B 0,C 180,E1 20424.178,E2 20424.178} C_VEL
LIN {X 0,Y 424.067,Z 778.23,A -85,B 0,C 180,E1 20421.593,E2 20421.593} C_VEL
LIN {X 0,Y 424.278,Z 772.086,A -85,B 0,C 180,E1 20418.994,E2 20418.994} C_VEL
LIN {X 0,Y 424.681,Z 764.479,A -85,B 0,C 180,E1 20416.496,E2 20416.496} C_VEL
LIN {X 0,Y 425.338,Z 755.162,A -85,B 0,C 180,E1 20414.035,E2 20414.035} C_VEL
LIN {X 0,Y 426.241,Z 744.275,A -85,B 0,C 180,E1 20411.678,E2 20411.678} C_VEL
LIN {X 0,Y 427.382,Z 732.017,A -85,B 0,C 180,E1 20409.455,E2 20409.455} C_VEL
LIN {X 0,Y 428.859,Z 717.422,A -85,B 0,C 180,E1 20407.23,E2 20407.23} C_VEL
LIN {X 0,Y 430.461,Z 702.036,A -85,B 0,C 180,E1 20405.257,E2 20405.257} C_VEL
LIN {X 0,Y 432.176,Z 685.587,A -85,B 0,C 180,E1 20403.478,E2 20403.478} C_VEL
LIN {X 0,Y 433.919,Z 668.028,A -85,B 0,C 180,E1 20401.885,E2 20401.885} C_VEL
LIN {X 0,Y 435.735,Z 648.669,A -85,B 0,C 180,E1 20400.438,E2 20400.438} C_VEL
LIN {X 0,Y 437.446,Z 628.182,A -85,B 0,C 180,E1 20399.202,E2 20399.202} C_VEL
LIN {X 0,Y 438.907,Z 608.019,A -85,B 0,C 180,E1 20398.248,E2 20398.248} C_VEL
LIN {X 0,Y 440.238,Z 585.612,A -85,B 0,C 180,E1 20397.462,E2 20397.462} C_VEL
LIN {X 0,Y 441.154,Z 562.58,A -85,B 0,C 180,E1 20396.924,E2 20396.924} C_VEL
LIN {X 0,Y 443.749,Z 480.887,A -85,B 0,C 180,E1 20395.284,E2 20395.284} C_VEL
LIN {X 0,Y 447.564,Z 402.285,A -85,B 0,C 180,E1 20393.51,E2 20393.51} C_VEL
LIN {X 0,Y 451.283,Z 344.071,A -85,B 0,C 180,E1 20392.054,E2 20392.054} C_VEL
LIN {X 0,Y 450.626,Z 334.976,A -85,B 0,C 180,E1 20391.635,E2 20391.635} C_VEL
LIN {X 0,Y 446.314,Z 326.182,A -85,B 0,C 180,E1 20390.563,E2 20390.563} C_VEL
LIN {X 0,Y 445.424,Z 324.189,A -85,B 0,C 180,E1 20390.226,E2 20390.226} C_VEL
LIN {X 0,Y 443.689,Z 318.701,A -85,B 0,C 180,E1 20388.822,E2 20388.822} C_VEL
LIN {X 0,Y 442.253,Z 314.227,A -85,B 0,C 180,E1 20387.287,E2 20387.287} C_VEL
LIN {X 0,Y 441.053,Z 311.15,A -85,B 0,C 180,E1 20385.35,E2 20385.35} C_VEL
LIN {X 0,Y 440.811,Z 310.485,A -85,B 0,C 180,E1 20384.134,E2 20384.134} C_VEL
LIN {X 0,Y 440.882,Z 310.923,A -85,B 0,C 180,E1 20382.871,E2 20382.871} C_VEL
LIN {X 0,Y 441.75,Z 313.755,A -85,B 0,C 180,E1 20380.853,E2 20380.853} C_VEL
LIN {X 0,Y 443.04,Z 317.992,A -85,B 0,C 180,E1 20379.191,E2 20379.191} C_VEL
LIN {X 0,Y 444.853,Z 323.959,A -85,B 0,C 180,E1 20377.494,E2 20377.494} C_VEL
LIN {X 0,Y 446.887,Z 332.274,A -85,B 0,C 180,E1 20375.69,E2 20375.69} C_VEL
LIN {X 0,Y 447.136,Z 333.991,A -85,B 0,C 180,E1 20375.391,E2 20375.391} C_VEL
LIN {X 0,Y 446.755,Z 337.38,A -85,B 0,C 180,E1 20375.043,E2 20375.043} C_VEL
LIN {X 0,Y 448.918,Z 357.315,A -85,B 0,C 180,E1 20373.813,E2 20373.813} C_VEL
LIN {X 0,Y 449.97,Z 371.91,A -85,B 0,C 180,E1 20373.104,E2 20373.104} C_VEL
LIN {X 0,Y 444.104,Z 453.902,A -85,B 0,C 180,E1 20371.035,E2 20371.035} C_VEL
LIN {X 0,Y 440.323,Z 530.109,A -85,B 0,C 180,E1 20369.26,E2 20369.26} C_VEL
LIN {X 0,Y 438.743,Z 567.556,A -85,B 0,C 180,E1 20368.39,E2 20368.39} C_VEL
LIN {X 0,Y 437.528,Z 588.027,A -85,B 0,C 180,E1 20367.663,E2 20367.663} C_VEL
LIN {X 0,Y 436.175,Z 606.498,A -85,B 0,C 180,E1 20366.772,E2 20366.772} C_VEL
LIN {X 0,Y 434.621,Z 625.027,A -85,B 0,C 180,E1 20365.626,E2 20365.626} C_VEL
LIN {X 0,Y 432.97,Z 642.58,A -85,B 0,C 180,E1 20364.271,E2 20364.271} C_VEL
LIN {X 0,Y 431.256,Z 659.501,A -85,B 0,C 180,E1 20362.666,E2 20362.666} C_VEL
LIN {X 0,Y 429.585,Z 675.07,A -85,B 0,C 180,E1 20360.861,E2 20360.861} C_VEL
LIN {X 0,Y 428.106,Z 688.808,A -85,B 0,C 180,E1 20358.932,E2 20358.932} C_VEL
LIN {X 0,Y 426.843,Z 700.897,A -85,B 0,C 180,E1 20356.885,E2 20356.885} C_VEL
LIN {X 0,Y 425.79,Z 711.738,A -85,B 0,C 180,E1 20354.65,E2 20354.65} C_VEL
LIN {X 0,Y 425.022,Z 720.736,A -85,B 0,C 180,E1 20352.361,E2 20352.361} C_VEL
LIN {X 0,Y 424.515,Z 728.003,A -85,B 0,C 180,E1 20350.037,E2 20350.037} C_VEL
LIN {X 0,Y 424.193,Z 733.833,A -85,B 0,C 180,E1 20347.585,E2 20347.585} C_VEL
LIN {X 0,Y 424.04,Z 738.089,A -85,B 0,C 180,E1 20345.005,E2 20345.005} C_VEL
LIN {X 0,Y 423.981,Z 740.549,A -85,B 0,C 180,E1 20342.432,E2 20342.432} C_VEL
LIN {X 0,Y 423.974,Z 741.282,A -85,B 0,C 180,E1 20339.864,E2 20339.864} C_VEL
LIN {X 0,Y 423.978,Z 740.303,A -85,B 0,C 180,E1 20337.296,E2 20337.296} C_VEL
LIN {X 0,Y 424.03,Z 737.598,A -85,B 0,C 180,E1 20334.723,E2 20334.723} C_VEL
LIN {X 0,Y 424.181,Z 733.087,A -85,B 0,C 180,E1 20332.142,E2 20332.142} C_VEL
LIN {X 0,Y 424.504,Z 727.048,A -85,B 0,C 180,E1 20329.688,E2 20329.688} C_VEL
LIN {X 0,Y 425.064,Z 719.102,A -85,B 0,C 180,E1 20327.225,E2 20327.225} C_VEL
LIN {X 0,Y 425.885,Z 709.625,A -85,B 0,C 180,E1 20324.894,E2 20324.894} C_VEL
LIN {X 0,Y 426.969,Z 698.661,A -85,B 0,C 180,E1 20322.698,E2 20322.698} C_VEL
LIN {X 0,Y 428.299,Z 686.217,A -85,B 0,C 180,E1 20320.64,E2 20320.64} C_VEL
LIN {X 0,Y 429.837,Z 672.239,A -85,B 0,C 180,E1 20318.722,E2 20318.722} C_VEL
LIN {X 0,Y 431.475,Z 657.269,A -85,B 0,C 180,E1 20317.016,E2 20317.016} C_VEL
LIN {X 0,Y 433.135,Z 641.442,A -85,B 0,C 180,E1 20315.52,E2 20315.52} C_VEL
LIN {X 0,Y 434.813,Z 624.151,A -85,B 0,C 180,E1 20314.185,E2 20314.185} C_VEL
LIN {X 0,Y 436.322,Z 606.476,A -85,B 0,C 180,E1 20313.09,E2 20313.09} C_VEL
LIN {X 0,Y 437.7,Z 587.49,A -85,B 0,C 180,E1 20312.182,E2 20312.182} C_VEL
LIN {X 0,Y 438.784,Z 568.171,A -85,B 0,C 180,E1 20311.512,E2 20311.512} C_VEL
LIN {X 0,Y 439.595,Z 546.054,A -85,B 0,C 180,E1 20311.017,E2 20311.017} C_VEL
LIN {X 0,Y 444.663,Z 368.932,A -85,B 0,C 180,E1 20307.637,E2 20307.637} C_VEL
LIN {X 0,Y 440.269,Z 340.137,A -85,B 0,C 180,E1 20306.583,E2 20306.583} C_VEL
LIN {X 0,Y 441.449,Z 327.276,A -85,B 0,C 180,E1 20305.305,E2 20305.305} C_VEL
LIN {X 0,Y 434.932,Z 308.602,A -85,B 0,C 180,E1 20302.633,E2 20302.633} C_VEL
LIN {X 0,Y 427.944,Z 290.418,A -85,B 0,C 180,E1 20299.82,E2 20299.82} C_VEL
LIN {X 0,Y 425.351,Z 283.703,A -85,B 0,C 180,E1 20298.692,E2 20298.692} C_VEL
LIN {X 0,Y 425.319,Z 283.506,A -85,B 0,C 180,E1 20294.851,E2 20294.851} C_VEL
LIN {X 0,Y 425.316,Z 283.507,A -85,B 0,C 180,E1 20290.988,E2 20290.988} C_VEL
LIN {X 0,Y 425.314,Z 283.508,A -85,B 0,C 180,E1 20287.16,E2 20287.16} C_VEL
LIN {X 0,Y 425.314,Z 283.507,A -85,B 0,C 180,E1 20283.375,E2 20283.375} C_VEL
LIN {X 0,Y 425.317,Z 283.497,A -85,B 0,C 180,E1 20280.422,E2 20280.422} C_VEL
LIN {X 0,Y 424.374,Z 283.608,A -85,B 0,C 180,E1 20279.384,E2 20279.384} C_VEL
LIN {X 0,Y 417.836,Z 284.436,A -85,B 0,C 180,E1 20276.386,E2 20276.386} C_VEL
LIN {X 0,Y 417.374,Z 284.482,A -85,B 0,C 180,E1 20275.698,E2 20275.698} C_VEL
LIN {X 0,Y 417.379,Z 284.483,A -85,B 0,C 180,E1 20271.798,E2 20271.798} C_VEL
LIN {X 0,Y 417.376,Z 284.484,A -85,B 0,C 180,E1 20268,E2 20268} C_VEL
LIN {X 0,Y 417.378,Z 284.754,A -85,B 0,C 180,E1 20266.617,E2 20266.617} C_VEL
LIN {X 0,Y 425.129,Z 305.321,A -85,B 0,C 180,E1 20263.882,E2 20263.882} C_VEL
LIN {X 0,Y 431.201,Z 323.769,A -85,B 0,C 180,E1 20261.64,E2 20261.64} C_VEL
LIN {X 0,Y 430.107,Z 353.014,A -85,B 0,C 180,E1 20259.003,E2 20259.003} C_VEL
LIN {X 0,Y 428.203,Z 394.572,A -85,B 0,C 180,E1 20255.293,E2 20255.293} C_VEL
LIN {X 0,Y 426.075,Z 438.721,A -85,B 0,C 180,E1 20251.346,E2 20251.346} C_VEL
LIN {X 0,Y 424.417,Z 478.081,A -85,B 0,C 180,E1 20247.875,E2 20247.875} C_VEL
LIN {X 0,Y 426.023,Z 493.695,A -85,B 0,C 180,E1 20247.498,E2 20247.498} C_VEL
LIN {X 0,Y 424.056,Z 621.138,A -85,B 0,C 180,E1 20245.276,E2 20245.276} C_VEL
LIN {X 0,Y 423.552,Z 637.168,A -85,B 0,C 180,E1 20244.749,E2 20244.749} C_VEL
LIN {X 0,Y 422.779,Z 653.135,A -85,B 0,C 180,E1 20243.961,E2 20243.961} C_VEL
LIN {X 0,Y 421.859,Z 667.544,A -85,B 0,C 180,E1 20242.99,E2 20242.99} C_VEL
LIN {X 0,Y 420.769,Z 681.882,A -85,B 0,C 180,E1 20241.736,E2 20241.736} C_VEL
LIN {X 0,Y 419.719,Z 694.525,A -85,B 0,C 180,E1 20240.333,E2 20240.333} C_VEL
LIN {X 0,Y 418.693,Z 706.205,A -85,B 0,C 180,E1 20238.709,E2 20238.709} C_VEL
LIN {X 0,Y 417.798,Z 716.532,A -85,B 0,C 180,E1 20236.913,E2 20236.913} C_VEL
LIN {X 0,Y 417.048,Z 725.79,A -85,B 0,C 180,E1 20234.853,E2 20234.853} C_VEL
LIN {X 0,Y 416.556,Z 732.803,A -85,B 0,C 180,E1 20232.81,E2 20232.81} C_VEL
LIN {X 0,Y 416.249,Z 738.236,A -85,B 0,C 180,E1 20230.643,E2 20230.643} C_VEL
LIN {X 0,Y 416.1,Z 741.901,A -85,B 0,C 180,E1 20228.426,E2 20228.426} C_VEL
LIN {X 0,Y 416.044,Z 743.855,A -85,B 0,C 180,E1 20226.039,E2 20226.039} C_VEL
LIN {X 0,Y 416.046,Z 743.917,A -85,B 0,C 180,E1 20223.911,E2 20223.911} C_VEL
LIN {X 0,Y 416.104,Z 742.138,A -85,B 0,C 180,E1 20221.579,E2 20221.579} C_VEL
LIN {X 0,Y 416.254,Z 738.717,A -85,B 0,C 180,E1 20219.389,E2 20219.389} C_VEL
LIN {X 0,Y 416.571,Z 733.245,A -85,B 0,C 180,E1 20217.149,E2 20217.149} C_VEL
LIN {X 0,Y 417.081,Z 726.26,A -85,B 0,C 180,E1 20215.073,E2 20215.073} C_VEL
LIN {X 0,Y 417.824,Z 717.355,A -85,B 0,C 180,E1 20213.061,E2 20213.061} C_VEL
LIN {X 0,Y 418.721,Z 707.313,A -85,B 0,C 180,E1 20211.274,E2 20211.274} C_VEL
LIN {X 0,Y 419.836,Z 694.926,A -85,B 0,C 180,E1 20209.532,E2 20209.532} C_VEL
LIN {X 0,Y 420.905,Z 682.328,A -85,B 0,C 180,E1 20208.127,E2 20208.127} C_VEL
LIN {X 0,Y 422.007,Z 667.978,A -85,B 0,C 180,E1 20206.866,E2 20206.866} C_VEL
LIN {X 0,Y 422.954,Z 653.486,A -85,B 0,C 180,E1 20205.89,E2 20205.89} C_VEL
LIN {X 0,Y 423.753,Z 636.992,A -85,B 0,C 180,E1 20205.078,E2 20205.078} C_VEL
LIN {X 0,Y 424.229,Z 620.962,A -85,B 0,C 180,E1 20204.562,E2 20204.562} C_VEL
LIN {X 0,Y 426.104,Z 490.472,A -85,B 0,C 180,E1 20202.261,E2 20202.261} C_VEL
LIN {X 0,Y 424.681,Z 478.164,A -85,B 0,C 180,E1 20201.931,E2 20201.931} C_VEL
LIN {X 0,Y 426.483,Z 435.275,A -85,B 0,C 180,E1 20198.153,E2 20198.153} C_VEL
LIN {X 0,Y 428.431,Z 392.366,A -85,B 0,C 180,E1 20194.387,E2 20194.387} C_VEL
LIN {X 0,Y 430.038,Z 351.813,A -85,B 0,C 180,E1 20190.85,E2 20190.85} C_VEL
LIN {X 0,Y 430.942,Z 322.307,A -85,B 0,C 180,E1 20188.25,E2 20188.25} C_VEL
LIN {X 0,Y 424.84,Z 303.788,A -85,B 0,C 180,E1 20186.036,E2 20186.036} C_VEL
LIN {X 0,Y 418.52,Z 287.76,A -85,B 0,C 180,E1 20183.963,E2 20183.963} C_VEL
LIN {X 0,Y 417.417,Z 284.724,A -85,B 0,C 180,E1 20183.498,E2 20183.498} C_VEL
LIN {X 0,Y 417.371,Z 284.498,A -85,B 0,C 180,E1 20179.742,E2 20179.742} C_VEL
LIN {X 0,Y 417.353,Z 284.492,A -85,B 0,C 180,E1 20175.993,E2 20175.993} C_VEL
LIN {X 0,Y 417.345,Z 284.499,A -85,B 0,C 180,E1 20172.196,E2 20172.196} C_VEL
LIN {X 0,Y 417.344,Z 284.496,A -85,B 0,C 180,E1 20168.345,E2 20168.345} C_VEL
LIN {X 0,Y 417.348,Z 284.496,A -85,B 0,C 180,E1 20164.535,E2 20164.535} C_VEL
LIN {X 0,Y 417.356,Z 284.496,A -85,B 0,C 180,E1 20160.687,E2 20160.687} C_VEL
LIN {X 0,Y 417.365,Z 284.493,A -85,B 0,C 180,E1 20156.842,E2 20156.842} C_VEL
LIN {X 0,Y 417.386,Z 284.49,A -85,B 0,C 180,E1 20152.983,E2 20152.983} C_VEL
LIN {X 0,Y 417.381,Z 284.495,A -85,B 0,C 180,E1 20149.092,E2 20149.092} C_VEL
LIN {X 0,Y 417.386,Z 284.491,A -85,B 0,C 180,E1 20145.149,E2 20145.149} C_VEL
LIN {X 0,Y 417.379,Z 284.491,A -85,B 0,C 180,E1 20141.277,E2 20141.277} C_VEL
LIN {X 0,Y 417.37,Z 284.492,A -85,B 0,C 180,E1 20137.462,E2 20137.462} C_VEL
LIN {X 0,Y 417.359,Z 284.499,A -85,B 0,C 180,E1 20133.63,E2 20133.63} C_VEL
LIN {X 0,Y 417.354,Z 284.494,A -85,B 0,C 180,E1 20129.861,E2 20129.861} C_VEL
LIN {X 0,Y 417.353,Z 284.495,A -85,B 0,C 180,E1 20125.984,E2 20125.984} C_VEL
LIN {X 0,Y 417.359,Z 284.494,A -85,B 0,C 180,E1 20122.172,E2 20122.172} C_VEL
LIN {X 0,Y 417.37,Z 284.495,A -85,B 0,C 180,E1 20118.365,E2 20118.365} C_VEL
LIN {X 0,Y 417.412,Z 284.728,A -85,B 0,C 180,E1 20114.985,E2 20114.985} C_VEL
LIN {X 0,Y 420.168,Z 291.543,A -85,B 0,C 180,E1 20113.86,E2 20113.86} C_VEL
LIN {X 0,Y 429.114,Z 312.779,A -85,B 0,C 180,E1 20110.674,E2 20110.674} C_VEL
LIN {X 0,Y 431.606,Z 318.766,A -85,B 0,C 180,E1 20109.882,E2 20109.882} C_VEL
LIN {X 0,Y 441.707,Z 337.509,A -85,B 0,C 180,E1 20108.499,E2 20108.499} C_VEL
LIN {X 0,Y 442.806,Z 347.412,A -85,B 0,C 180,E1 20108.175,E2 20108.175} C_VEL
LIN {X 0,Y 436.724,Z 537.254,A -85,B 0,C 180,E1 20104.531,E2 20104.531} C_VEL
LIN {X 0,Y 435.415,Z 578.599,A -85,B 0,C 180,E1 20103.713,E2 20103.713} C_VEL
LIN {X 0,Y 434.193,Z 599.455,A -85,B 0,C 180,E1 20103.075,E2 20103.075} C_VEL
LIN {X 0,Y 432.594,Z 620.027,A -85,B 0,C 180,E1 20102.198,E2 20102.198} C_VEL
LIN {X 0,Y 430.742,Z 640.166,A -85,B 0,C 180,E1 20101.07,E2 20101.07} C_VEL
LIN {X 0,Y 428.785,Z 658.638,A -85,B 0,C 180,E1 20099.779,E2 20099.779} C_VEL
LIN {X 0,Y 426.722,Z 676.673,A -85,B 0,C 180,E1 20098.247,E2 20098.247} C_VEL
LIN {X 0,Y 424.692,Z 693.464,A -85,B 0,C 180,E1 20096.538,E2 20096.538} C_VEL
LIN {X 0,Y 422.633,Z 709.984,A -85,B 0,C 180,E1 20094.53,E2 20094.53} C_VEL
LIN {X 0,Y 420.895,Z 724.267,A -85,B 0,C 180,E1 20092.469,E2 20092.469} C_VEL
LIN {X 0,Y 419.364,Z 737.445,A -85,B 0,C 180,E1 20090.223,E2 20090.223} C_VEL
LIN {X 0,Y 418.11,Z 749.237,A -85,B 0,C 180,E1 20087.822,E2 20087.822} C_VEL
LIN {X 0,Y 417.166,Z 759.532,A -85,B 0,C 180,E1 20085.285,E2 20085.285} C_VEL
LIN {X 0,Y 416.539,Z 767.912,A -85,B 0,C 180,E1 20082.756,E2 20082.756} C_VEL
LIN {X 0,Y 416.163,Z 775.241,A -85,B 0,C 180,E1 20079.96,E2 20079.96} C_VEL
LIN {X 0,Y 415.997,Z 780.424,A -85,B 0,C 180,E1 20077.317,E2 20077.317} C_VEL
LIN {X 0,Y 415.961,Z 783.972,A -85,B 0,C 180,E1 20074.686,E2 20074.686} C_VEL
LIN {X 0,Y 415.97,Z 785.865,A -85,B 0,C 180,E1 20072.065,E2 20072.065} C_VEL
LIN {X 0,Y 415.974,Z 786.226,A -85,B 0,C 180,E1 20069.31,E2 20069.31} C_VEL
LIN {X 0,Y 415.965,Z 785.009,A -85,B 0,C 180,E1 20066.691,E2 20066.691} C_VEL
LIN {X 0,Y 415.988,Z 782.19,A -85,B 0,C 180,E1 20064.066,E2 20064.066} C_VEL
LIN {X 0,Y 416.077,Z 777.698,A -85,B 0,C 180,E1 20061.43,E2 20061.43} C_VEL
LIN {X 0,Y 416.298,Z 771.492,A -85,B 0,C 180,E1 20058.781,E2 20058.781} C_VEL
LIN {X 0,Y 416.729,Z 763.9,A -85,B 0,C 180,E1 20056.258,E2 20056.258} C_VEL
LIN {X 0,Y 417.438,Z 754.436,A -85,B 0,C 180,E1 20053.724,E2 20053.724} C_VEL
LIN {X 0,Y 418.479,Z 742.779,A -85,B 0,C 180,E1 20051.181,E2 20051.181} C_VEL
LIN {X 0,Y 419.723,Z 730.288,A -85,B 0,C 180,E1 20048.916,E2 20048.916} C_VEL
LIN {X 0,Y 421.277,Z 715.819,A -85,B 0,C 180,E1 20046.708,E2 20046.708} C_VEL
LIN {X 0,Y 423.02,Z 699.925,A -85,B 0,C 180,E1 20044.67,E2 20044.67} C_VEL
LIN {X 0,Y 424.947,Z 682.47,A -85,B 0,C 180,E1 20042.797,E2 20042.797} C_VEL
LIN {X 0,Y 426.872,Z 663.986,A -85,B 0,C 180,E1 20041.149,E2 20041.149} C_VEL
LIN {X 0,Y 428.718,Z 644.913,A -85,B 0,C 180,E1 20039.75,E2 20039.75} C_VEL
LIN {X 0,Y 430.474,Z 625.001,A -85,B 0,C 180,E1 20038.57,E2 20038.57} C_VEL
LIN {X 0,Y 432.01,Z 604.551,A -85,B 0,C 180,E1 20037.617,E2 20037.617} C_VEL
LIN {X 0,Y 433.366,Z 583.279,A -85,B 0,C 180,E1 20036.886,E2 20036.886} C_VEL
LIN {X 0,Y 434.335,Z 560.012,A -85,B 0,C 180,E1 20036.34,E2 20036.34} C_VEL
LIN {X 0,Y 437.202,Z 482.276,A -85,B 0,C 180,E1 20034.703,E2 20034.703} C_VEL
LIN {X 0,Y 441.361,Z 407.179,A -85,B 0,C 180,E1 20032.928,E2 20032.928} C_VEL
LIN {X 0,Y 445.911,Z 345.782,A -85,B 0,C 180,E1 20031.325,E2 20031.325} C_VEL
LIN {X 0,Y 445.566,Z 338.925,A -85,B 0,C 180,E1 20030.985,E2 20030.985} C_VEL
LIN {X 0,Y 441.709,Z 330.881,A -85,B 0,C 180,E1 20029.915,E2 20029.915} C_VEL
LIN {X 0,Y 439.019,Z 325.909,A -85,B 0,C 180,E1 20029.01,E2 20029.01} C_VEL
LIN {X 0,Y 437.703,Z 322.033,A -85,B 0,C 180,E1 20027.741,E2 20027.741} C_VEL
LIN {X 0,Y 436.917,Z 319.704,A -85,B 0,C 180,E1 20026.695,E2 20026.695} C_VEL
LIN {X 0,Y 436.257,Z 317.093,A -85,B 0,C 180,E1 20024.717,E2 20024.717} C_VEL
LIN {X 0,Y 436.162,Z 317.206,A -85,B 0,C 180,E1 20023.089,E2 20023.089} C_VEL
LIN {X 0,Y 436.83,Z 320.025,A -85,B 0,C 180,E1 20020.944,E2 20020.944} C_VEL
LIN {X 0,Y 437.947,Z 324.346,A -85,B 0,C 180,E1 20019.227,E2 20019.227} C_VEL
LIN {X 0,Y 439.622,Z 330.524,A -85,B 0,C 180,E1 20017.461,E2 20017.461} C_VEL
LIN {X 0,Y 440.842,Z 335.919,A -85,B 0,C 180,E1 20016.263,E2 20016.263} C_VEL
LIN {X 0,Y 441.837,Z 339.013,A -85,B 0,C 180,E1 20015.881,E2 20015.881} C_VEL
LIN {X 0,Y 443.51,Z 357.592,A -85,B 0,C 180,E1 20014.654,E2 20014.654} C_VEL
LIN {X 0,Y 444.469,Z 373.275,A -85,B 0,C 180,E1 20013.832,E2 20013.832} C_VEL
LIN {X 0,Y 438.012,Z 452.967,A -85,B 0,C 180,E1 20011.727,E2 20011.727} C_VEL
LIN {X 0,Y 433.8,Z 526.459,A -85,B 0,C 180,E1 20009.922,E2 20009.922} C_VEL
LIN {X 0,Y 431.85,Z 567.574,A -85,B 0,C 180,E1 20008.928,E2 20008.928} C_VEL
LIN {X 0,Y 430.518,Z 588.238,A -85,B 0,C 180,E1 20008.176,E2 20008.176} C_VEL
LIN {X 0,Y 429.047,Z 606.93,A -85,B 0,C 180,E1 20007.253,E2 20007.253} C_VEL
LIN {X 0,Y 427.395,Z 625.318,A -85,B 0,C 180,E1 20006.091,E2 20006.091} C_VEL
LIN {X 0,Y 425.637,Z 642.814,A -85,B 0,C 180,E1 20004.717,E2 20004.717} C_VEL
LIN {X 0,Y 423.921,Z 658.661,A -85,B 0,C 180,E1 20003.196,E2 20003.196} C_VEL
LIN {X 0,Y 422.223,Z 673.664,A -85,B 0,C 180,E1 20001.461,E2 20001.461} C_VEL
LIN {X 0,Y 420.671,Z 687.19,A -85,B 0,C 180,E1 19999.58,E2 19999.58} C_VEL
LIN {X 0,Y 419.25,Z 699.883,A -85,B 0,C 180,E1 19997.453,E2 19997.453} C_VEL
LIN {X 0,Y 418.111,Z 710.679,A -85,B 0,C 180,E1 19995.251,E2 19995.251} C_VEL
LIN {X 0,Y 417.224,Z 720.135,A -85,B 0,C 180,E1 19992.877,E2 19992.877} C_VEL
LIN {X 0,Y 416.607,Z 728.023,A -85,B 0,C 180,E1 19990.369,E2 19990.369} C_VEL
LIN {X 0,Y 416.233,Z 734.25,A -85,B 0,C 180,E1 19987.73,E2 19987.73} C_VEL
LIN {X 0,Y 416.062,Z 738.522,A -85,B 0,C 180,E1 19985.101,E2 19985.101} C_VEL
LIN {X 0,Y 415.995,Z 740.986,A -85,B 0,C 180,E1 19982.479,E2 19982.479} C_VEL
LIN {X 0,Y 415.986,Z 741.71,A -85,B 0,C 180,E1 19979.862,E2 19979.862} C_VEL
LIN {X 0,Y 415.991,Z 740.711,A -85,B 0,C 180,E1 19977.244,E2 19977.244} C_VEL
LIN {X 0,Y 416.048,Z 737.973,A -85,B 0,C 180,E1 19974.621,E2 19974.621} C_VEL
LIN {X 0,Y 416.215,Z 733.417,A -85,B 0,C 180,E1 19971.99,E2 19971.99} C_VEL
LIN {X 0,Y 416.566,Z 727.326,A -85,B 0,C 180,E1 19969.489,E2 19969.489} C_VEL
LIN {X 0,Y 417.173,Z 719.314,A -85,B 0,C 180,E1 19966.979,E2 19966.979} C_VEL
LIN {X 0,Y 418.06,Z 709.762,A -85,B 0,C 180,E1 19964.604,E2 19964.604} C_VEL
LIN {X 0,Y 419.218,Z 698.715,A -85,B 0,C 180,E1 19962.367,E2 19962.367} C_VEL
LIN {X 0,Y 420.635,Z 686.186,A -85,B 0,C 180,E1 19960.273,E2 19960.273} C_VEL
LIN {X 0,Y 422.266,Z 672.107,A -85,B 0,C 180,E1 19958.322,E2 19958.322} C_VEL
LIN {X 0,Y 424.004,Z 656.944,A -85,B 0,C 180,E1 19956.58,E2 19956.58} C_VEL
LIN {X 0,Y 425.752,Z 640.958,A -85,B 0,C 180,E1 19955.06,E2 19955.06} C_VEL
LIN {X 0,Y 427.445,Z 624.321,A -85,B 0,C 180,E1 19953.761,E2 19953.761} C_VEL
LIN {X 0,Y 429.05,Z 606.308,A -85,B 0,C 180,E1 19952.632,E2 19952.632} C_VEL
LIN {X 0,Y 430.482,Z 587.36,A -85,B 0,C 180,E1 19951.717,E2 19951.717} C_VEL
LIN {X 0,Y 431.624,Z 568.015,A -85,B 0,C 180,E1 19951.038,E2 19951.038} C_VEL
LIN {X 0,Y 432.473,Z 545.888,A -85,B 0,C 180,E1 19950.534,E2 19950.534} C_VEL
LIN {X 0,Y 437.927,Z 370.277,A -85,B 0,C 180,E1 19947.097,E2 19947.097} C_VEL
LIN {X 0,Y 433.368,Z 339.946,A -85,B 0,C 180,E1 19945.962,E2 19945.962} C_VEL
LIN {X 0,Y 434.241,Z 329.996,A -85,B 0,C 180,E1 19944.953,E2 19944.953} C_VEL
LIN {X 0,Y 428.031,Z 312.209,A -85,B 0,C 180,E1 19942.364,E2 19942.364} C_VEL
LIN {X 0,Y 420.921,Z 293.897,A -85,B 0,C 180,E1 19939.477,E2 19939.477} C_VEL
LIN {X 0,Y 417.386,Z 284.693,A -85,B 0,C 180,E1 19937.917,E2 19937.917} C_VEL
LIN {X 0,Y 417.37,Z 284.496,A -85,B 0,C 180,E1 19934.198,E2 19934.198} C_VEL
LIN {X 0,Y 417.38,Z 284.495,A -85,B 0,C 180,E1 19930.302,E2 19930.302} C_VEL
LIN {X 0,Y 417.378,Z 284.492,A -85,B 0,C 180,E1 19926.397,E2 19926.397} C_VEL
LIN {X 0,Y 417.377,Z 284.492,A -85,B 0,C 180,E1 19922.454,E2 19922.454} C_VEL
LIN {X 0,Y 417.364,Z 284.482,A -85,B 0,C 180,E1 19918.63,E2 19918.63} C_VEL
LIN {X 0,Y 417.374,Z 284.482,A -85,B 0,C 180,E1 19915.698,E2 19915.698} C_VEL
LIN {X 0,Y 416.355,Z 284.611,A -85,B 0,C 180,E1 19914.64,E2 19914.64} C_VEL
LIN {X 0,Y 409.833,Z 285.422,A -85,B 0,C 180,E1 19911.584,E2 19911.584} C_VEL
LIN {X 0,Y 409.404,Z 285.475,A -85,B 0,C 180,E1 19910.883,E2 19910.883} C_VEL
LIN {X 0,Y 409.424,Z 285.654,A -85,B 0,C 180,E1 19907.335,E2 19907.335} C_VEL
LIN {X 0,Y 409.945,Z 287.565,A -85,B 0,C 180,E1 19907.02,E2 19907.02} C_VEL
LIN {X 0,Y 416.426,Z 303.82,A -85,B 0,C 180,E1 19904.817,E2 19904.817} C_VEL
LIN {X 0,Y 423.283,Z 324.023,A -85,B 0,C 180,E1 19902.276,E2 19902.276} C_VEL
LIN {X 0,Y 424.155,Z 327.905,A -85,B 0,C 180,E1 19901.836,E2 19901.836} C_VEL
LIN {X 0,Y 422.202,Z 369.171,A -85,B 0,C 180,E1 19898.102,E2 19898.102} C_VEL
LIN {X 0,Y 420.196,Z 409.88,A -85,B 0,C 180,E1 19894.437,E2 19894.437} C_VEL
LIN {X 0,Y 418.12,Z 452.276,A -85,B 0,C 180,E1 19890.618,E2 19890.618} C_VEL
LIN {X 0,Y 416.97,Z 478.502,A -85,B 0,C 180,E1 19888.295,E2 19888.295} C_VEL
LIN {X 0,Y 418.618,Z 494.474,A -85,B 0,C 180,E1 19887.901,E2 19887.901} C_VEL
LIN {X 0,Y 416.535,Z 621.551,A -85,B 0,C 180,E1 19885.644,E2 19885.644} C_VEL
LIN {X 0,Y 416.005,Z 637.569,A -85,B 0,C 180,E1 19885.107,E2 19885.107} C_VEL
LIN {X 0,Y 415.223,Z 653.003,A -85,B 0,C 180,E1 19884.336,E2 19884.336} C_VEL
LIN {X 0,Y 414.257,Z 667.567,A -85,B 0,C 180,E1 19883.349,E2 19883.349} C_VEL
LIN {X 0,Y 413.107,Z 681.979,A -85,B 0,C 180,E1 19882.072,E2 19882.072} C_VEL
LIN {X 0,Y 411.997,Z 694.7,A -85,B 0,C 180,E1 19880.644,E2 19880.644} C_VEL
LIN {X 0,Y 410.863,Z 706.887,A -85,B 0,C 180,E1 19878.918,E2 19878.918} C_VEL
LIN {X 0,Y 409.96,Z 716.704,A -85,B 0,C 180,E1 19877.179,E2 19877.179} C_VEL
LIN {X 0,Y 409.167,Z 725.785,A -85,B 0,C 180,E1 19875.134,E2 19875.134} C_VEL
LIN {X 0,Y 408.633,Z 732.854,A -85,B 0,C 180,E1 19873.074,E2 19873.074} C_VEL
LIN {X 0,Y 408.288,Z 738.413,A -85,B 0,C 180,E1 19870.845,E2 19870.845} C_VEL
LIN {X 0,Y 408.118,Z 742.175,A -85,B 0,C 180,E1 19868.589,E2 19868.589} C_VEL
LIN {X 0,Y 408.055,Z 744.119,A -85,B 0,C 180,E1 19866.308,E2 19866.308} C_VEL
LIN {X 0,Y 408.056,Z 744.351,A -85,B 0,C 180,E1 19863.987,E2 19863.987} C_VEL
LIN {X 0,Y 408.114,Z 742.658,A -85,B 0,C 180,E1 19861.624,E2 19861.624} C_VEL
LIN {X 0,Y 408.274,Z 739.319,A -85,B 0,C 180,E1 19859.379,E2 19859.379} C_VEL
LIN {X 0,Y 408.578,Z 734.395,A -85,B 0,C 180,E1 19857.263,E2 19857.263} C_VEL
LIN {X 0,Y 409.107,Z 727.572,A -85,B 0,C 180,E1 19855.12,E2 19855.12} C_VEL
LIN {X 0,Y 409.847,Z 719.188,A -85,B 0,C 180,E1 19853.123,E2 19853.123} C_VEL
LIN {X 0,Y 410.777,Z 709.377,A -85,B 0,C 180,E1 19851.28,E2 19851.28} C_VEL
LIN {X 0,Y 411.856,Z 698.132,A -85,B 0,C 180,E1 19849.597,E2 19849.597} C_VEL
LIN {X 0,Y 413.017,Z 685.395,A -85,B 0,C 180,E1 19848.078,E2 19848.078} C_VEL
LIN {X 0,Y 414.138,Z 672.032,A -85,B 0,C 180,E1 19846.814,E2 19846.814} C_VEL
LIN {X 0,Y 415.226,Z 656.9,A -85,B 0,C 180,E1 19845.711,E2 19845.711} C_VEL
LIN {X 0,Y 416.072,Z 641.531,A -85,B 0,C 180,E1 19844.88,E2 19844.88} C_VEL
LIN {X 0,Y 416.686,Z 624.56,A -85,B 0,C 180,E1 19844.259,E2 19844.259} C_VEL
LIN {X 0,Y 417.094,Z 601.073,A -85,B 0,C 180,E1 19843.788,E2 19843.788} C_VEL
LIN {X 0,Y 418.77,Z 491.392,A -85,B 0,C 180,E1 19841.841,E2 19841.841} C_VEL
LIN {X 0,Y 417.272,Z 478.572,A -85,B 0,C 180,E1 19841.495,E2 19841.495} C_VEL
LIN {X 0,Y 419.22,Z 435.152,A -85,B 0,C 180,E1 19837.632,E2 19837.632} C_VEL
LIN {X 0,Y 421.374,Z 390.604,A -85,B 0,C 180,E1 19833.672,E2 19833.672} C_VEL
LIN {X 0,Y 423.186,Z 346.815,A -85,B 0,C 180,E1 19829.825,E2 19829.825} C_VEL
LIN {X 0,Y 423.888,Z 325.31,A -85,B 0,C 180,E1 19827.919,E2 19827.919} C_VEL
LIN {X 0,Y 417.839,Z 306.895,A -85,B 0,C 180,E1 19825.666,E2 19825.666} C_VEL
LIN {X 0,Y 410.798,Z 289.054,A -85,B 0,C 180,E1 19823.299,E2 19823.299} C_VEL
LIN {X 0,Y 409.445,Z 285.747,A -85,B 0,C 180,E1 19822.772,E2 19822.772} C_VEL
LIN {X 0,Y 409.441,Z 285.48,A -85,B 0,C 180,E1 19819.398,E2 19819.398} C_VEL
LIN {X 0,Y 409.445,Z 285.474,A -85,B 0,C 180,E1 19815.437,E2 19815.437} C_VEL
LIN {X 0,Y 409.438,Z 285.488,A -85,B 0,C 180,E1 19811.552,E2 19811.552} C_VEL
LIN {X 0,Y 409.44,Z 285.487,A -85,B 0,C 180,E1 19807.578,E2 19807.578} C_VEL
LIN {X 0,Y 409.43,Z 285.483,A -85,B 0,C 180,E1 19803.641,E2 19803.641} C_VEL
LIN {X 0,Y 409.426,Z 285.486,A -85,B 0,C 180,E1 19799.721,E2 19799.721} C_VEL
LIN {X 0,Y 409.418,Z 285.482,A -85,B 0,C 180,E1 19795.799,E2 19795.799} C_VEL
LIN {X 0,Y 409.41,Z 285.486,A -85,B 0,C 180,E1 19791.999,E2 19791.999} C_VEL
LIN {X 0,Y 409.409,Z 285.486,A -85,B 0,C 180,E1 19788.162,E2 19788.162} C_VEL
LIN {X 0,Y 409.409,Z 285.48,A -85,B 0,C 180,E1 19784.194,E2 19784.194} C_VEL
LIN {X 0,Y 409.414,Z 285.483,A -85,B 0,C 180,E1 19780.305,E2 19780.305} C_VEL
LIN {X 0,Y 409.42,Z 285.484,A -85,B 0,C 180,E1 19776.39,E2 19776.39} C_VEL
LIN {X 0,Y 409.429,Z 285.481,A -85,B 0,C 180,E1 19772.513,E2 19772.513} C_VEL
LIN {X 0,Y 409.44,Z 285.481,A -85,B 0,C 180,E1 19768.658,E2 19768.658} C_VEL
LIN {X 0,Y 409.442,Z 285.484,A -85,B 0,C 180,E1 19764.809,E2 19764.809} C_VEL
LIN {X 0,Y 409.447,Z 285.483,A -85,B 0,C 180,E1 19760.942,E2 19760.942} C_VEL
LIN {X 0,Y 409.441,Z 285.482,A -85,B 0,C 180,E1 19757.054,E2 19757.054} C_VEL
LIN {X 0,Y 409.455,Z 285.752,A -85,B 0,C 180,E1 19755.81,E2 19755.81} C_VEL
LIN {X 0,Y 413.697,Z 295.947,A -85,B 0,C 180,E1 19754.109,E2 19754.109} C_VEL
LIN {X 0,Y 422.584,Z 317.111,A -85,B 0,C 180,E1 19750.892,E2 19750.892} C_VEL
LIN {X 0,Y 423.974,Z 319.962,A -85,B 0,C 180,E1 19750.592,E2 19750.592} C_VEL
LIN {X 0,Y 435.36,Z 340.774,A -85,B 0,C 180,E1 19749,E2 19749} C_VEL
LIN {X 0,Y 436.163,Z 348.636,A -85,B 0,C 180,E1 19748.743,E2 19748.743} C_VEL
LIN {X 0,Y 429.865,Z 532.714,A -85,B 0,C 180,E1 19745.133,E2 19745.133} C_VEL
LIN {X 0,Y 428.331,Z 578.448,A -85,B 0,C 180,E1 19744.211,E2 19744.211} C_VEL
LIN {X 0,Y 427.043,Z 599.463,A -85,B 0,C 180,E1 19743.556,E2 19743.556} C_VEL
LIN {X 0,Y 425.338,Z 620.362,A -85,B 0,C 180,E1 19742.647,E2 19742.647} C_VEL
LIN {X 0,Y 423.343,Z 641.074,A -85,B 0,C 180,E1 19741.462,E2 19741.462} C_VEL
LIN {X 0,Y 421.182,Z 660.578,A -85,B 0,C 180,E1 19740.057,E2 19740.057} C_VEL
LIN {X 0,Y 418.95,Z 678.998,A -85,B 0,C 180,E1 19738.43,E2 19738.43} C_VEL
LIN {X 0,Y 416.812,Z 695.719,A -85,B 0,C 180,E1 19736.651,E2 19736.651} C_VEL
LIN {X 0,Y 414.743,Z 711.551,A -85,B 0,C 180,E1 19734.648,E2 19734.648} C_VEL
LIN {X 0,Y 412.908,Z 725.909,A -85,B 0,C 180,E1 19732.493,E2 19732.493} C_VEL
LIN {X 0,Y 411.253,Z 739.579,A -85,B 0,C 180,E1 19730.046,E2 19730.046} C_VEL
LIN {X 0,Y 409.975,Z 751.287,A -85,B 0,C 180,E1 19727.527,E2 19727.527} C_VEL
LIN {X 0,Y 409.08,Z 760.974,A -85,B 0,C 180,E1 19725.014,E2 19725.014} C_VEL
LIN {X 0,Y 408.457,Z 769.464,A -85,B 0,C 180,E1 19722.295,E2 19722.295} C_VEL
LIN {X 0,Y 408.127,Z 776.005,A -85,B 0,C 180,E1 19719.588,E2 19719.588} C_VEL
LIN {X 0,Y 408.001,Z 780.825,A -85,B 0,C 180,E1 19716.895,E2 19716.895} C_VEL
LIN {X 0,Y 407.975,Z 784.153,A -85,B 0,C 180,E1 19714.074,E2 19714.074} C_VEL
LIN {X 0,Y 407.977,Z 785.727,A -85,B 0,C 180,E1 19711.403,E2 19711.403} C_VEL
LIN {X 0,Y 407.987,Z 785.708,A -85,B 0,C 180,E1 19708.875,E2 19708.875} C_VEL
LIN {X 0,Y 407.981,Z 784.184,A -85,B 0,C 180,E1 19706.204,E2 19706.204} C_VEL
LIN {X 0,Y 408,Z 781.107,A -85,B 0,C 180,E1 19703.526,E2 19703.526} C_VEL
LIN {X 0,Y 408.103,Z 776.347,A -85,B 0,C 180,E1 19700.835,E2 19700.835} C_VEL
LIN {X 0,Y 408.363,Z 770.157,A -85,B 0,C 180,E1 19698.273,E2 19698.273} C_VEL
LIN {X 0,Y 408.894,Z 761.726,A -85,B 0,C 180,E1 19695.54,E2 19695.54} C_VEL
LIN {X 0,Y 409.7,Z 751.884,A -85,B 0,C 180,E1 19692.97,E2 19692.97} C_VEL
LIN {X 0,Y 410.808,Z 740.532,A -85,B 0,C 180,E1 19690.521,E2 19690.521} C_VEL
LIN {X 0,Y 412.193,Z 727.752,A -85,B 0,C 180,E1 19688.213,E2 19688.213} C_VEL
LIN {X 0,Y 413.956,Z 712.453,A -85,B 0,C 180,E1 19685.907,E2 19685.907} C_VEL
LIN {X 0,Y 415.898,Z 695.878,A -85,B 0,C 180,E1 19683.821,E2 19683.821} C_VEL
LIN {X 0,Y 417.908,Z 678.404,A -85,B 0,C 180,E1 19681.987,E2 19681.987} C_VEL
LIN {X 0,Y 419.918,Z 660.099,A -85,B 0,C 180,E1 19680.39,E2 19680.39} C_VEL
LIN {X 0,Y 421.825,Z 641.387,A -85,B 0,C 180,E1 19679.044,E2 19679.044} C_VEL
LIN {X 0,Y 423.642,Z 621.478,A -85,B 0,C 180,E1 19677.884,E2 19677.884} C_VEL
LIN {X 0,Y 425.313,Z 600.478,A -85,B 0,C 180,E1 19676.931,E2 19676.931} C_VEL
LIN {X 0,Y 426.713,Z 578.887,A -85,B 0,C 180,E1 19676.215,E2 19676.215} C_VEL
LIN {X 0,Y 428.431,Z 536.993,A -85,B 0,C 180,E1 19675.282,E2 19675.282} C_VEL
LIN {X 0,Y 431.798,Z 465.751,A -85,B 0,C 180,E1 19673.655,E2 19673.655} C_VEL
LIN {X 0,Y 436.632,Z 395.58,A -85,B 0,C 180,E1 19671.876,E2 19671.876} C_VEL
LIN {X 0,Y 440.822,Z 347.159,A -85,B 0,C 180,E1 19670.538,E2 19670.538} C_VEL
LIN {X 0,Y 440.653,Z 343.03,A -85,B 0,C 180,E1 19670.307,E2 19670.307} C_VEL
LIN {X 0,Y 437.475,Z 336.184,A -85,B 0,C 180,E1 19669.307,E2 19669.307} C_VEL
LIN {X 0,Y 434.845,Z 331.426,A -85,B 0,C 180,E1 19668.354,E2 19668.354} C_VEL
LIN {X 0,Y 432.59,Z 327.549,A -85,B 0,C 180,E1 19667.307,E2 19667.307} C_VEL
LIN {X 0,Y 431.952,Z 325.727,A -85,B 0,C 180,E1 19666.385,E2 19666.385} C_VEL
LIN {X 0,Y 431.536,Z 323.543,A -85,B 0,C 180,E1 19664.591,E2 19664.591} C_VEL
LIN {X 0,Y 431.432,Z 323.706,A -85,B 0,C 180,E1 19663.11,E2 19663.11} C_VEL
LIN {X 0,Y 431.955,Z 326.581,A -85,B 0,C 180,E1 19660.924,E2 19660.924} C_VEL
LIN {X 0,Y 433.064,Z 331.226,A -85,B 0,C 180,E1 19659.072,E2 19659.072} C_VEL
LIN {X 0,Y 434.094,Z 335.275,A -85,B 0,C 180,E1 19657.95,E2 19657.95} C_VEL
LIN {X 0,Y 437.443,Z 343.141,A -85,B 0,C 180,E1 19656.568,E2 19656.568} C_VEL
LIN {X 0,Y 438.732,Z 362.342,A -85,B 0,C 180,E1 19655.27,E2 19655.27} C_VEL
LIN {X 0,Y 439.181,Z 375.076,A -85,B 0,C 180,E1 19654.587,E2 19654.587} C_VEL
LIN {X 0,Y 432.067,Z 453.004,A -85,B 0,C 180,E1 19652.437,E2 19652.437} C_VEL
LIN {X 0,Y 427.349,Z 524.988,A -85,B 0,C 180,E1 19650.576,E2 19650.576} C_VEL
LIN {X 0,Y 425.041,Z 568.087,A -85,B 0,C 180,E1 19649.486,E2 19649.486} C_VEL
LIN {X 0,Y 423.582,Z 588.718,A -85,B 0,C 180,E1 19648.708,E2 19648.708} C_VEL
LIN {X 0,Y 421.977,Z 607.641,A -85,B 0,C 180,E1 19647.749,E2 19647.749} C_VEL
LIN {X 0,Y 420.222,Z 625.834,A -85,B 0,C 180,E1 19646.571,E2 19646.571} C_VEL
LIN {X 0,Y 418.356,Z 643.232,A -85,B 0,C 180,E1 19645.176,E2 19645.176} C_VEL
LIN {X 0,Y 416.456,Z 659.71,A -85,B 0,C 180,E1 19643.562,E2 19643.562} C_VEL
LIN {X 0,Y 414.595,Z 675.147,A -85,B 0,C 180,E1 19641.727,E2 19641.727} C_VEL
LIN {X 0,Y 412.85,Z 689.394,A -85,B 0,C 180,E1 19639.672,E2 19639.672} C_VEL
LIN {X 0,Y 411.39,Z 701.591,A -85,B 0,C 180,E1 19637.54,E2 19637.54} C_VEL
LIN {X 0,Y 410.189,Z 712.307,A -85,B 0,C 180,E1 19635.263,E2 19635.263} C_VEL
LIN {X 0,Y 409.272,Z 721.526,A -85,B 0,C 180,E1 19632.845,E2 19632.845} C_VEL
LIN {X 0,Y 408.634,Z 729.185,A -85,B 0,C 180,E1 19630.289,E2 19630.289} C_VEL
LIN {X 0,Y 408.26,Z 734.944,A -85,B 0,C 180,E1 19627.741,E2 19627.741} C_VEL
LIN {X 0,Y 408.085,Z 738.969,A -85,B 0,C 180,E1 19625.201,E2 19625.201} C_VEL
LIN {X 0,Y 408.009,Z 741.429,A -85,B 0,C 180,E1 19622.528,E2 19622.528} C_VEL
LIN {X 0,Y 407.997,Z 742.14,A -85,B 0,C 180,E1 19619.859,E2 19619.859} C_VEL
LIN {X 0,Y 408.003,Z 741.115,A -85,B 0,C 180,E1 19617.19,E2 19617.19} C_VEL
LIN {X 0,Y 408.067,Z 738.34,A -85,B 0,C 180,E1 19614.516,E2 19614.516} C_VEL
LIN {X 0,Y 408.239,Z 734.039,A -85,B 0,C 180,E1 19611.975,E2 19611.975} C_VEL
LIN {X 0,Y 408.607,Z 727.988,A -85,B 0,C 180,E1 19609.424,E2 19609.424} C_VEL
LIN {X 0,Y 409.246,Z 720.031,A -85,B 0,C 180,E1 19606.866,E2 19606.866} C_VEL
LIN {X 0,Y 410.177,Z 710.522,A -85,B 0,C 180,E1 19604.446,E2 19604.446} C_VEL
LIN {X 0,Y 411.391,Z 699.517,A -85,B 0,C 180,E1 19602.167,E2 19602.167} C_VEL
LIN {X 0,Y 412.919,Z 686.635,A -85,B 0,C 180,E1 19599.973,E2 19599.973} C_VEL
LIN {X 0,Y 414.575,Z 673.027,A -85,B 0,C 180,E1 19598.048,E2 19598.048} C_VEL
LIN {X 0,Y 416.382,Z 658.041,A -85,B 0,C 180,E1 19596.282,E2 19596.282} C_VEL
LIN {X 0,Y 418.203,Z 642.211,A -85,B 0,C 180,E1 19594.737,E2 19594.737} C_VEL
LIN {X 0,Y 420.071,Z 624.636,A -85,B 0,C 180,E1 19593.338,E2 19593.338} C_VEL
LIN {X 0,Y 421.795,Z 606.079,A -85,B 0,C 180,E1 19592.161,E2 19592.161} C_VEL
LIN {X 0,Y 423.294,Z 587.005,A -85,B 0,C 180,E1 19591.231,E2 19591.231} C_VEL
LIN {X 0,Y 424.503,Z 567.385,A -85,B 0,C 180,E1 19590.538,E2 19590.538} C_VEL
LIN {X 0,Y 425.458,Z 542.817,A -85,B 0,C 180,E1 19589.981,E2 19589.981} C_VEL
LIN {X 0,Y 431.126,Z 371.276,A -85,B 0,C 180,E1 19586.54,E2 19586.54} C_VEL
LIN {X 0,Y 426.483,Z 339.985,A -85,B 0,C 180,E1 19585.347,E2 19585.347} C_VEL
LIN {X 0,Y 427.084,Z 332.903,A -85,B 0,C 180,E1 19584.626,E2 19584.626} C_VEL
LIN {X 0,Y 420.829,Z 314.961,A -85,B 0,C 180,E1 19581.965,E2 19581.965} C_VEL
LIN {X 0,Y 413.241,Z 295.326,A -85,B 0,C 180,E1 19578.807,E2 19578.807} C_VEL
LIN {X 0,Y 409.469,Z 285.685,A -85,B 0,C 180,E1 19577.111,E2 19577.111} C_VEL
LIN {X 0,Y 409.437,Z 285.476,A -85,B 0,C 180,E1 19573.303,E2 19573.303} C_VEL
LIN {X 0,Y 409.444,Z 285.483,A -85,B 0,C 180,E1 19569.415,E2 19569.415} C_VEL
LIN {X 0,Y 409.438,Z 285.487,A -85,B 0,C 180,E1 19565.536,E2 19565.536} C_VEL
LIN {X 0,Y 409.443,Z 285.486,A -85,B 0,C 180,E1 19561.672,E2 19561.672} C_VEL
LIN {X 0,Y 409.443,Z 285.478,A -85,B 0,C 180,E1 19557.804,E2 19557.804} C_VEL
LIN {X 0,Y 409.444,Z 285.474,A -85,B 0,C 180,E1 19553.916,E2 19553.916} C_VEL
LIN {X 0,Y 409.404,Z 285.475,A -85,B 0,C 180,E1 19550.883,E2 19550.883} C_VEL
LIN {X 0,Y 408.633,Z 286.013,A -85,B 0,C 180,E1 19549.833,E2 19549.833} C_VEL
LIN {X 0,Y 406.513,Z 288.248,A -85,B 0,C 180,E1 19548.529,E2 19548.529} C_VEL
LIN {X 0,Y 405.109,Z 291.765,A -85,B 0,C 180,E1 19547.458,E2 19547.458} C_VEL
LIN {X 0,Y 405.189,Z 295.467,A -85,B 0,C 180,E1 19546.743,E2 19546.743} C_VEL
LIN {X 0,Y 405.561,Z 296.905,A -85,B 0,C 180,E1 19546.535,E2 19546.535} C_VEL
LIN {X 0,Y 412.964,Z 317.049,A -85,B 0,C 180,E1 19543.855,E2 19543.855} C_VEL
LIN {X 0,Y 417.029,Z 329.886,A -85,B 0,C 180,E1 19542.252,E2 19542.252} C_VEL
LIN {X 0,Y 414.96,Z 371.575,A -85,B 0,C 180,E1 19538.453,E2 19538.453} C_VEL
LIN {X 0,Y 412.836,Z 411.688,A -85,B 0,C 180,E1 19534.794,E2 19534.794} C_VEL
LIN {X 0,Y 410.672,Z 454.282,A -85,B 0,C 180,E1 19530.928,E2 19530.928} C_VEL
LIN {X 0,Y 409.505,Z 478.654,A -85,B 0,C 180,E1 19528.734,E2 19528.734} C_VEL
LIN {X 0,Y 411.224,Z 495.271,A -85,B 0,C 180,E1 19528.315,E2 19528.315} C_VEL
LIN {X 0,Y 409.029,Z 621.938,A -85,B 0,C 180,E1 19526.024,E2 19526.024} C_VEL
LIN {X 0,Y 408.474,Z 637.95,A -85,B 0,C 180,E1 19525.478,E2 19525.478} C_VEL
LIN {X 0,Y 407.614,Z 654.079,A -85,B 0,C 180,E1 19524.653,E2 19524.653} C_VEL
LIN {X 0,Y 406.598,Z 668.45,A -85,B 0,C 180,E1 19523.648,E2 19523.648} C_VEL
LIN {X 0,Y 405.397,Z 682.78,A -85,B 0,C 180,E1 19522.348,E2 19522.348} C_VEL
LIN {X 0,Y 404.228,Z 695.407,A -85,B 0,C 180,E1 19520.893,E2 19520.893} C_VEL
LIN {X 0,Y 403.037,Z 707.547,A -85,B 0,C 180,E1 19519.134,E2 19519.134} C_VEL
LIN {X 0,Y 402.083,Z 717.305,A -85,B 0,C 180,E1 19517.361,E2 19517.361} C_VEL
LIN {X 0,Y 401.228,Z 726.581,A -85,B 0,C 180,E1 19515.219,E2 19515.219} C_VEL
LIN {X 0,Y 400.68,Z 733.373,A -85,B 0,C 180,E1 19513.176,E2 19513.176} C_VEL
LIN {X 0,Y 400.312,Z 738.903,A -85,B 0,C 180,E1 19510.903,E2 19510.903} C_VEL
LIN {X 0,Y 400.132,Z 742.614,A -85,B 0,C 180,E1 19508.605,E2 19508.605} C_VEL
LIN {X 0,Y 400.064,Z 744.585,A -85,B 0,C 180,E1 19506.168,E2 19506.168} C_VEL
LIN {X 0,Y 400.066,Z 744.723,A -85,B 0,C 180,E1 19503.907,E2 19503.907} C_VEL
LIN {X 0,Y 400.134,Z 742.993,A -85,B 0,C 180,E1 19501.495,E2 19501.495} C_VEL
LIN {X 0,Y 400.315,Z 739.607,A -85,B 0,C 180,E1 19499.204,E2 19499.204} C_VEL
LIN {X 0,Y 400.683,Z 734.177,A -85,B 0,C 180,E1 19496.876,E2 19496.876} C_VEL
LIN {X 0,Y 401.239,Z 727.638,A -85,B 0,C 180,E1 19494.822,E2 19494.822} C_VEL
LIN {X 0,Y 402.072,Z 718.864,A -85,B 0,C 180,E1 19492.729,E2 19492.729} C_VEL
LIN {X 0,Y 403.085,Z 708.931,A -85,B 0,C 180,E1 19490.857,E2 19490.857} C_VEL
LIN {X 0,Y 404.242,Z 697.485,A -85,B 0,C 180,E1 19489.152,E2 19489.152} C_VEL
LIN {X 0,Y 405.505,Z 684.436,A -85,B 0,C 180,E1 19487.596,E2 19487.596} C_VEL
LIN {X 0,Y 406.721,Z 670.306,A -85,B 0,C 180,E1 19486.283,E2 19486.283} C_VEL
LIN {X 0,Y 407.821,Z 655.569,A -85,B 0,C 180,E1 19485.223,E2 19485.223} C_VEL
LIN {X 0,Y 408.703,Z 639.406,A -85,B 0,C 180,E1 19484.379,E2 19484.379} C_VEL
LIN {X 0,Y 409.283,Z 623.246,A -85,B 0,C 180,E1 19483.81,E2 19483.81} C_VEL
LIN {X 0,Y 410.285,Z 565.115,A -85,B 0,C 180,E1 19482.729,E2 19482.729} C_VEL
LIN {X 0,Y 411.454,Z 492.273,A -85,B 0,C 180,E1 19481.404,E2 19481.404} C_VEL
LIN {X 0,Y 409.896,Z 478.596,A -85,B 0,C 180,E1 19481.009,E2 19481.009} C_VEL
LIN {X 0,Y 411.938,Z 436.084,A -85,B 0,C 180,E1 19477.185,E2 19477.185} C_VEL
LIN {X 0,Y 413.964,Z 395.766,A -85,B 0,C 180,E1 19473.581,E2 19473.581} C_VEL
LIN {X 0,Y 415.691,Z 358.54,A -85,B 0,C 180,E1 19470.26,E2 19470.26} C_VEL
LIN {X 0,Y 416.909,Z 328.405,A -85,B 0,C 180,E1 19467.573,E2 19467.573} C_VEL
LIN {X 0,Y 411.048,Z 310.536,A -85,B 0,C 180,E1 19465.349,E2 19465.349} C_VEL
LIN {X 0,Y 404.238,Z 293.317,A -85,B 0,C 180,E1 19463.005,E2 19463.005} C_VEL
LIN {X 0,Y 401.548,Z 286.939,A -85,B 0,C 180,E1 19462.048,E2 19462.048} C_VEL
LIN {X 0,Y 401.507,Z 286.466,A -85,B 0,C 180,E1 19461.627,E2 19461.627} C_VEL
LIN {X 0,Y 401.494,Z 286.468,A -85,B 0,C 180,E1 19457.688,E2 19457.688} C_VEL
LIN {X 0,Y 401.49,Z 286.478,A -85,B 0,C 180,E1 19453.783,E2 19453.783} C_VEL
LIN {X 0,Y 401.479,Z 286.477,A -85,B 0,C 180,E1 19449.895,E2 19449.895} C_VEL
LIN {X 0,Y 401.475,Z 286.473,A -85,B 0,C 180,E1 19446.005,E2 19446.005} C_VEL
LIN {X 0,Y 401.468,Z 286.477,A -85,B 0,C 180,E1 19442.141,E2 19442.141} C_VEL
LIN {X 0,Y 401.468,Z 286.472,A -85,B 0,C 180,E1 19438.288,E2 19438.288} C_VEL
LIN {X 0,Y 401.469,Z 286.475,A -85,B 0,C 180,E1 19434.283,E2 19434.283} C_VEL
LIN {X 0,Y 401.473,Z 286.469,A -85,B 0,C 180,E1 19430.395,E2 19430.395} C_VEL
LIN {X 0,Y 401.477,Z 286.472,A -85,B 0,C 180,E1 19426.462,E2 19426.462} C_VEL
LIN {X 0,Y 401.488,Z 286.473,A -85,B 0,C 180,E1 19422.612,E2 19422.612} C_VEL
LIN {X 0,Y 401.493,Z 286.468,A -85,B 0,C 180,E1 19418.646,E2 19418.646} C_VEL
LIN {X 0,Y 401.496,Z 286.472,A -85,B 0,C 180,E1 19414.682,E2 19414.682} C_VEL
LIN {X 0,Y 401.509,Z 286.468,A -85,B 0,C 180,E1 19410.785,E2 19410.785} C_VEL
LIN {X 0,Y 401.502,Z 286.472,A -85,B 0,C 180,E1 19406.78,E2 19406.78} C_VEL
LIN {X 0,Y 401.504,Z 286.472,A -85,B 0,C 180,E1 19402.762,E2 19402.762} C_VEL
LIN {X 0,Y 401.508,Z 286.47,A -85,B 0,C 180,E1 19398.766,E2 19398.766} C_VEL
LIN {X 0,Y 401.541,Z 286.736,A -85,B 0,C 180,E1 19396.664,E2 19396.664} C_VEL
LIN {X 0,Y 404.51,Z 293.868,A -85,B 0,C 180,E1 19395.414,E2 19395.414} C_VEL
LIN {X 0,Y 413.46,Z 315.115,A -85,B 0,C 180,E1 19392.054,E2 19392.054} C_VEL
LIN {X 0,Y 415.177,Z 319.194,A -85,B 0,C 180,E1 19391.499,E2 19391.499} C_VEL
LIN {X 0,Y 428.834,Z 343.693,A -85,B 0,C 180,E1 19389.542,E2 19389.542} C_VEL
LIN {X 0,Y 429.555,Z 349.719,A -85,B 0,C 180,E1 19389.329,E2 19389.329} C_VEL
LIN {X 0,Y 422.825,Z 534.371,A -85,B 0,C 180,E1 19385.626,E2 19385.626} C_VEL
LIN {X 0,Y 421.256,Z 578.403,A -85,B 0,C 180,E1 19384.718,E2 19384.718} C_VEL
LIN {X 0,Y 419.91,Z 599.404,A -85,B 0,C 180,E1 19384.05,E2 19384.05} C_VEL
LIN {X 0,Y 418.113,Z 620.428,A -85,B 0,C 180,E1 19383.12,E2 19383.12} C_VEL
LIN {X 0,Y 416.039,Z 641.087,A -85,B 0,C 180,E1 19381.917,E2 19381.917} C_VEL
LIN {X 0,Y 413.78,Z 660.538,A -85,B 0,C 180,E1 19380.492,E2 19380.492} C_VEL
LIN {X 0,Y 411.454,Z 678.932,A -85,B 0,C 180,E1 19378.838,E2 19378.838} C_VEL
LIN {X 0,Y 409.219,Z 695.653,A -85,B 0,C 180,E1 19377.028,E2 19377.028} C_VEL
LIN {X 0,Y 407.127,Z 710.957,A -85,B 0,C 180,E1 19375.063,E2 19375.063} C_VEL
LIN {X 0,Y 405.255,Z 724.947,A -85,B 0,C 180,E1 19372.941,E2 19372.941} C_VEL
LIN {X 0,Y 403.582,Z 738.014,A -85,B 0,C 180,E1 19370.595,E2 19370.595} C_VEL
LIN {X 0,Y 402.229,Z 749.671,A -85,B 0,C 180,E1 19368.101,E2 19368.101} C_VEL
LIN {X 0,Y 401.216,Z 759.861,A -85,B 0,C 180,E1 19365.463,E2 19365.463} C_VEL
LIN {X 0,Y 400.52,Z 768.473,A -85,B 0,C 180,E1 19362.689,E2 19362.689} C_VEL
LIN {X 0,Y 400.173,Z 774.86,A -85,B 0,C 180,E1 19360.071,E2 19360.071} C_VEL
LIN {X 0,Y 400.004,Z 779.926,A -85,B 0,C 180,E1 19357.322,E2 19357.322} C_VEL
LIN {X 0,Y 399.977,Z 783.361,A -85,B 0,C 180,E1 19354.587,E2 19354.587} C_VEL
LIN {X 0,Y 399.99,Z 785.136,A -85,B 0,C 180,E1 19351.861,E2 19351.861} C_VEL
LIN {X 0,Y 400.001,Z 785.331,A -85,B 0,C 180,E1 19349.139,E2 19349.139} C_VEL
LIN {X 0,Y 399.986,Z 783.985,A -85,B 0,C 180,E1 19346.416,E2 19346.416} C_VEL
LIN {X 0,Y 400.003,Z 781.06,A -85,B 0,C 180,E1 19343.684,E2 19343.684} C_VEL
LIN {X 0,Y 400.1,Z 776.391,A -85,B 0,C 180,E1 19340.94,E2 19340.94} C_VEL
LIN {X 0,Y 400.375,Z 769.983,A -85,B 0,C 180,E1 19338.182,E2 19338.182} C_VEL
LIN {X 0,Y 400.935,Z 761.544,A -85,B 0,C 180,E1 19335.374,E2 19335.374} C_VEL
LIN {X 0,Y 401.776,Z 751.827,A -85,B 0,C 180,E1 19332.773,E2 19332.773} C_VEL
LIN {X 0,Y 402.944,Z 740.542,A -85,B 0,C 180,E1 19330.276,E2 19330.276} C_VEL
LIN {X 0,Y 404.402,Z 727.805,A -85,B 0,C 180,E1 19327.924,E2 19327.924} C_VEL
LIN {X 0,Y 406.132,Z 713.597,A -85,B 0,C 180,E1 19325.722,E2 19325.722} C_VEL
LIN {X 0,Y 408.074,Z 697.927,A -85,B 0,C 180,E1 19323.672,E2 19323.672} C_VEL
LIN {X 0,Y 410.113,Z 681.403,A -85,B 0,C 180,E1 19321.85,E2 19321.85} C_VEL
LIN {X 0,Y 412.357,Z 662.488,A -85,B 0,C 180,E1 19320.112,E2 19320.112} C_VEL
LIN {X 0,Y 414.568,Z 642.382,A -85,B 0,C 180,E1 19318.603,E2 19318.603} C_VEL
LIN {X 0,Y 416.592,Z 621.862,A -85,B 0,C 180,E1 19317.367,E2 19317.367} C_VEL
LIN {X 0,Y 418.438,Z 600.512,A -85,B 0,C 180,E1 19316.37,E2 19316.37} C_VEL
LIN {X 0,Y 419.994,Z 578.492,A -85,B 0,C 180,E1 19315.616,E2 19315.616} C_VEL
LIN {X 0,Y 424.81,Z 481.827,A -85,B 0,C 180,E1 19313.342,E2 19313.342} C_VEL
LIN {X 0,Y 429.849,Z 413.206,A -85,B 0,C 180,E1 19311.552,E2 19311.552} C_VEL
LIN {X 0,Y 436.14,Z 349.307,A -85,B 0,C 180,E1 19309.738,E2 19309.738} C_VEL
LIN {X 0,Y 436.039,Z 347.252,A -85,B 0,C 180,E1 19309.606,E2 19309.606} C_VEL
LIN {X 0,Y 433.189,Z 340.804,A -85,B 0,C 180,E1 19308.544,E2 19308.544} C_VEL
LIN {X 0,Y 430.212,Z 335.369,A -85,B 0,C 180,E1 19307.209,E2 19307.209} C_VEL
LIN {X 0,Y 428.633,Z 333.013,A -85,B 0,C 180,E1 19306.313,E2 19306.313} C_VEL
LIN {X 0,Y 427.038,Z 330.221,A -85,B 0,C 180,E1 19304.809,E2 19304.809} C_VEL
LIN {X 0,Y 426.718,Z 330.119,A -85,B 0,C 180,E1 19303.22,E2 19303.22} C_VEL
LIN {X 0,Y 427.103,Z 332.831,A -85,B 0,C 180,E1 19301.094,E2 19301.094} C_VEL
LIN {X 0,Y 428.732,Z 337.025,A -85,B 0,C 180,E1 19299.623,E2 19299.623} C_VEL
LIN {X 0,Y 431.191,Z 342.596,A -85,B 0,C 180,E1 19298.226,E2 19298.226} C_VEL
LIN {X 0,Y 433.391,Z 348.399,A -85,B 0,C 180,E1 19297.207,E2 19297.207} C_VEL
LIN {X 0,Y 434.095,Z 366.894,A -85,B 0,C 180,E1 19295.928,E2 19295.928} C_VEL
LIN {X 0,Y 434.18,Z 376.926,A -85,B 0,C 180,E1 19295.382,E2 19295.382} C_VEL
LIN {X 0,Y 426.359,Z 453.054,A -85,B 0,C 180,E1 19293.189,E2 19293.189} C_VEL
LIN {X 0,Y 421.045,Z 524.214,A -85,B 0,C 180,E1 19291.257,E2 19291.257} C_VEL
LIN {X 0,Y 418.334,Z 568.989,A -85,B 0,C 180,E1 19290.067,E2 19290.067} C_VEL
LIN {X 0,Y 416.746,Z 589.436,A -85,B 0,C 180,E1 19289.267,E2 19289.267} C_VEL
LIN {X 0,Y 414.927,Z 609.187,A -85,B 0,C 180,E1 19288.229,E2 19288.229} C_VEL
LIN {X 0,Y 412.905,Z 628.546,A -85,B 0,C 180,E1 19286.925,E2 19286.925} C_VEL
LIN {X 0,Y 410.899,Z 645.811,A -85,B 0,C 180,E1 19285.473,E2 19285.473} C_VEL
LIN {X 0,Y 408.864,Z 662.153,A -85,B 0,C 180,E1 19283.797,E2 19283.797} C_VEL
LIN {X 0,Y 406.908,Z 677.187,A -85,B 0,C 180,E1 19281.931,E2 19281.931} C_VEL
LIN {X 0,Y 405.129,Z 690.8,A -85,B 0,C 180,E1 19279.894,E2 19279.894} C_VEL
LIN {X 0,Y 403.603,Z 702.744,A -85,B 0,C 180,E1 19277.74,E2 19277.74} C_VEL
LIN {X 0,Y 402.335,Z 713.337,A -85,B 0,C 180,E1 19275.421,E2 19275.421} C_VEL
LIN {X 0,Y 401.364,Z 722.444,A -85,B 0,C 180,E1 19272.956,E2 19272.956} C_VEL
LIN {X 0,Y 400.714,Z 729.647,A -85,B 0,C 180,E1 19270.494,E2 19270.494} C_VEL
LIN {X 0,Y 400.306,Z 735.408,A -85,B 0,C 180,E1 19267.896,E2 19267.896} C_VEL
LIN {X 0,Y 400.109,Z 739.43,A -85,B 0,C 180,E1 19265.305,E2 19265.305} C_VEL
LIN {X 0,Y 400.024,Z 741.88,A -85,B 0,C 180,E1 19262.578,E2 19262.578} C_VEL
LIN {X 0,Y 400.01,Z 742.584,A -85,B 0,C 180,E1 19259.999,E2 19259.999} C_VEL
LIN {X 0,Y 400.014,Z 741.619,A -85,B 0,C 180,E1 19257.277,E2 19257.277} C_VEL
LIN {X 0,Y 400.081,Z 738.898,A -85,B 0,C 180,E1 19254.55,E2 19254.55} C_VEL
LIN {X 0,Y 400.275,Z 734.348,A -85,B 0,C 180,E1 19251.814,E2 19251.814} C_VEL
LIN {X 0,Y 400.673,Z 728.235,A -85,B 0,C 180,E1 19249.212,E2 19249.212} C_VEL
LIN {X 0,Y 401.363,Z 720.196,A -85,B 0,C 180,E1 19246.604,E2 19246.604} C_VEL
LIN {X 0,Y 402.36,Z 710.601,A -85,B 0,C 180,E1 19244.136,E2 19244.136} C_VEL
LIN {X 0,Y 403.655,Z 699.494,A -85,B 0,C 180,E1 19241.813,E2 19241.813} C_VEL
LIN {X 0,Y 405.226,Z 686.896,A -85,B 0,C 180,E1 19239.64,E2 19239.64} C_VEL
LIN {X 0,Y 407.024,Z 672.753,A -85,B 0,C 180,E1 19237.619,E2 19237.619} C_VEL
LIN {X 0,Y 408.929,Z 657.613,A -85,B 0,C 180,E1 19235.823,E2 19235.823} C_VEL
LIN {X 0,Y 410.907,Z 641.043,A -85,B 0,C 180,E1 19234.202,E2 19234.202} C_VEL
LIN {X 0,Y 412.803,Z 623.895,A -85,B 0,C 180,E1 19232.833,E2 19232.833} C_VEL
LIN {X 0,Y 414.534,Z 606.056,A -85,B 0,C 180,E1 19231.69,E2 19231.69} C_VEL
LIN {X 0,Y 416.106,Z 586.84,A -85,B 0,C 180,E1 19230.741,E2 19230.741} C_VEL
LIN {X 0,Y 417.393,Z 566.886,A -85,B 0,C 180,E1 19230.03,E2 19230.03} C_VEL
LIN {X 0,Y 418.498,Z 538.975,A -85,B 0,C 180,E1 19229.397,E2 19229.397} C_VEL
LIN {X 0,Y 424.371,Z 372.403,A -85,B 0,C 180,E1 19225.973,E2 19225.973} C_VEL
LIN {X 0,Y 419.632,Z 339.846,A -85,B 0,C 180,E1 19224.703,E2 19224.703} C_VEL
LIN {X 0,Y 419.936,Z 335.776,A -85,B 0,C 180,E1 19224.285,E2 19224.285} C_VEL
LIN {X 0,Y 413.636,Z 317.721,A -85,B 0,C 180,E1 19221.555,E2 19221.555} C_VEL
LIN {X 0,Y 406.443,Z 299.158,A -85,B 0,C 180,E1 19218.512,E2 19218.512} C_VEL
LIN {X 0,Y 401.52,Z 286.668,A -85,B 0,C 180,E1 19216.295,E2 19216.295} C_VEL
LIN {X 0,Y 401.5,Z 286.469,A -85,B 0,C 180,E1 19212.446,E2 19212.446} C_VEL
LIN {X 0,Y 401.505,Z 286.472,A -85,B 0,C 180,E1 19208.505,E2 19208.505} C_VEL
LIN {X 0,Y 401.499,Z 286.47,A -85,B 0,C 180,E1 19204.482,E2 19204.482} C_VEL
LIN {X 0,Y 401.497,Z 286.462,A -85,B 0,C 180,E1 19200.496,E2 19200.496} C_VEL
LIN {X 0,Y 401.484,Z 286.474,A -85,B 0,C 180,E1 19196.611,E2 19196.611} C_VEL
LIN {X 0,Y 401.476,Z 286.476,A -85,B 0,C 180,E1 19192.708,E2 19192.708} C_VEL
LIN {X 0,Y 401.462,Z 286.47,A -85,B 0,C 180,E1 19188.841,E2 19188.841} C_VEL
LIN {X 0,Y 401.541,Z 286.773,A -85,B 0,C 180,E1 19188.005,E2 19188.005} C_VEL
LIN {X 0,Y 404.764,Z 295.056,A -85,B 0,C 180,E1 19186.8,E2 19186.8} C_VEL
LIN {X 0,Y 405.561,Z 296.905,A -85,B 0,C 180,E1 19186.535,E2 19186.535} C_VEL
LIN {X 0,Y 406.594,Z 302.848,A -85,B 0,C 180,E1 19185.842,E2 19185.842} C_VEL
LIN {X 0,Y 406.744,Z 321.177,A -85,B 0,C 180,E1 19184.029,E2 19184.029} C_VEL
LIN {X 0,Y 407.641,Z 325.401,A -85,B 0,C 180,E1 19183.533,E2 19183.533} C_VEL
LIN {X 0,Y 409.893,Z 332.99,A -85,B 0,C 180,E1 19182.587,E2 19182.587} C_VEL
LIN {X 0,Y 407.639,Z 375.156,A -85,B 0,C 180,E1 19178.701,E2 19178.701} C_VEL
LIN {X 0,Y 405.431,Z 415.192,A -85,B 0,C 180,E1 19175.024,E2 19175.024} C_VEL
LIN {X 0,Y 403.186,Z 457.574,A -85,B 0,C 180,E1 19171.138,E2 19171.138} C_VEL
LIN {X 0,Y 402.086,Z 479.024,A -85,B 0,C 180,E1 19169.182,E2 19169.182} C_VEL
LIN {X 0,Y 403.84,Z 496.079,A -85,B 0,C 180,E1 19168.74,E2 19168.74} C_VEL
LIN {X 0,Y 401.543,Z 622.324,A -85,B 0,C 180,E1 19166.419,E2 19166.419} C_VEL
LIN {X 0,Y 400.96,Z 638.334,A -85,B 0,C 180,E1 19165.863,E2 19165.863} C_VEL
LIN {X 0,Y 400.091,Z 653.927,A -85,B 0,C 180,E1 19165.056,E2 19165.056} C_VEL
LIN {X 0,Y 399.033,Z 668.365,A -85,B 0,C 180,E1 19164.04,E2 19164.04} C_VEL
LIN {X 0,Y 397.76,Z 682.856,A -85,B 0,C 180,E1 19162.709,E2 19162.709} C_VEL
LIN {X 0,Y 396.552,Z 695.298,A -85,B 0,C 180,E1 19161.262,E2 19161.262} C_VEL
LIN {X 0,Y 395.31,Z 707.279,A -85,B 0,C 180,E1 19159.509,E2 19159.509} C_VEL
LIN {X 0,Y 394.288,Z 717.193,A -85,B 0,C 180,E1 19157.703,E2 19157.703} C_VEL
LIN {X 0,Y 393.375,Z 726.397,A -85,B 0,C 180,E1 19155.562,E2 19155.562} C_VEL
LIN {X 0,Y 392.762,Z 733.47,A -85,B 0,C 180,E1 19153.436,E2 19153.436} C_VEL
LIN {X 0,Y 392.355,Z 739.072,A -85,B 0,C 180,E1 19151.119,E2 19151.119} C_VEL
LIN {X 0,Y 392.153,Z 742.883,A -85,B 0,C 180,E1 19148.776,E2 19148.776} C_VEL
LIN {X 0,Y 392.075,Z 744.872,A -85,B 0,C 180,E1 19146.4,E2 19146.4} C_VEL
LIN {X 0,Y 392.076,Z 745.149,A -85,B 0,C 180,E1 19143.986,E2 19143.986} C_VEL
LIN {X 0,Y 392.141,Z 743.583,A -85,B 0,C 180,E1 19141.603,E2 19141.603} C_VEL
LIN {X 0,Y 392.336,Z 740.201,A -85,B 0,C 180,E1 19139.187,E2 19139.187} C_VEL
LIN {X 0,Y 392.707,Z 735.085,A -85,B 0,C 180,E1 19136.895,E2 19136.895} C_VEL
LIN {X 0,Y 393.319,Z 728.311,A -85,B 0,C 180,E1 19134.689,E2 19134.689} C_VEL
LIN {X 0,Y 394.141,Z 720.215,A -85,B 0,C 180,E1 19132.68,E2 19132.68} C_VEL
LIN {X 0,Y 395.214,Z 710.247,A -85,B 0,C 180,E1 19130.73,E2 19130.73} C_VEL
LIN {X 0,Y 396.4,Z 699.307,A -85,B 0,C 180,E1 19129.022,E2 19129.022} C_VEL
LIN {X 0,Y 397.775,Z 685.884,A -85,B 0,C 180,E1 19127.36,E2 19127.36} C_VEL
LIN {X 0,Y 399.025,Z 672.379,A -85,B 0,C 180,E1 19126.048,E2 19126.048} C_VEL
LIN {X 0,Y 400.251,Z 656.946,A -85,B 0,C 180,E1 19124.893,E2 19124.893} C_VEL
LIN {X 0,Y 401.169,Z 641.449,A -85,B 0,C 180,E1 19124.045,E2 19124.045} C_VEL
LIN {X 0,Y 401.832,Z 624.77,A -85,B 0,C 180,E1 19123.423,E2 19123.423} C_VEL
LIN {X 0,Y 402.409,Z 593.858,A -85,B 0,C 180,E1 19122.807,E2 19122.807} C_VEL
LIN {X 0,Y 404.148,Z 493.038,A -85,B 0,C 180,E1 19120.949,E2 19120.949} C_VEL
LIN {X 0,Y 402.544,Z 478.977,A -85,B 0,C 180,E1 19120.534,E2 19120.534} C_VEL
LIN {X 0,Y 404.689,Z 437.04,A -85,B 0,C 180,E1 19116.721,E2 19116.721} C_VEL
LIN {X 0,Y 407.087,Z 392.855,A -85,B 0,C 180,E1 19112.708,E2 19112.708} C_VEL
LIN {X 0,Y 409.144,Z 348.932,A -85,B 0,C 180,E1 19108.779,E2 19108.779} C_VEL
LIN {X 0,Y 409.823,Z 331.006,A -85,B 0,C 180,E1 19107.145,E2 19107.145} C_VEL
LIN {X 0,Y 403.97,Z 313.246,A -85,B 0,C 180,E1 19104.883,E2 19104.883} C_VEL
LIN {X 0,Y 396.828,Z 295.284,A -85,B 0,C 180,E1 19102.363,E2 19102.363} C_VEL
LIN {X 0,Y 393.6,Z 287.76,A -85,B 0,C 180,E1 19101.186,E2 19101.186} C_VEL
LIN {X 0,Y 393.563,Z 287.458,A -85,B 0,C 180,E1 19099.44,E2 19099.44} C_VEL
LIN {X 0,Y 393.566,Z 287.451,A -85,B 0,C 180,E1 19095.472,E2 19095.472} C_VEL
LIN {X 0,Y 393.561,Z 287.464,A -85,B 0,C 180,E1 19091.43,E2 19091.43} C_VEL
LIN {X 0,Y 393.57,Z 287.463,A -85,B 0,C 180,E1 19087.445,E2 19087.445} C_VEL
LIN {X 0,Y 393.561,Z 287.461,A -85,B 0,C 180,E1 19083.35,E2 19083.35} C_VEL
LIN {X 0,Y 393.569,Z 287.456,A -85,B 0,C 180,E1 19079.273,E2 19079.273} C_VEL
LIN {X 0,Y 393.564,Z 287.462,A -85,B 0,C 180,E1 19075.191,E2 19075.191} C_VEL
LIN {X 0,Y 393.566,Z 287.458,A -85,B 0,C 180,E1 19071.196,E2 19071.196} C_VEL
LIN {X 0,Y 393.564,Z 287.456,A -85,B 0,C 180,E1 19067.231,E2 19067.231} C_VEL
LIN {X 0,Y 393.562,Z 287.46,A -85,B 0,C 180,E1 19063.284,E2 19063.284} C_VEL
LIN {X 0,Y 393.566,Z 287.46,A -85,B 0,C 180,E1 19059.207,E2 19059.207} C_VEL
LIN {X 0,Y 393.562,Z 287.459,A -85,B 0,C 180,E1 19055.217,E2 19055.217} C_VEL
LIN {X 0,Y 393.572,Z 287.46,A -85,B 0,C 180,E1 19051.139,E2 19051.139} C_VEL
LIN {X 0,Y 393.559,Z 287.463,A -85,B 0,C 180,E1 19047.234,E2 19047.234} C_VEL
LIN {X 0,Y 393.553,Z 287.462,A -85,B 0,C 180,E1 19043.342,E2 19043.342} C_VEL
LIN {X 0,Y 393.55,Z 287.466,A -85,B 0,C 180,E1 19039.429,E2 19039.429} C_VEL
LIN {X 0,Y 393.582,Z 287.73,A -85,B 0,C 180,E1 19037.551,E2 19037.551} C_VEL
LIN {X 0,Y 402.202,Z 308.042,A -85,B 0,C 180,E1 19034.075,E2 19034.075} C_VEL
LIN {X 0,Y 406.944,Z 319.226,A -85,B 0,C 180,E1 19032.359,E2 19032.359} C_VEL
LIN {X 0,Y 422.36,Z 346.857,A -85,B 0,C 180,E1 19030.078,E2 19030.078} C_VEL
LIN {X 0,Y 422.986,Z 349.882,A -85,B 0,C 180,E1 19029.944,E2 19029.944} C_VEL
LIN {X 0,Y 415.677,Z 539.395,A -85,B 0,C 180,E1 19026.062,E2 19026.062} C_VEL
LIN {X 0,Y 414.165,Z 578.769,A -85,B 0,C 180,E1 19025.223,E2 19025.223} C_VEL
LIN {X 0,Y 412.749,Z 599.725,A -85,B 0,C 180,E1 19024.539,E2 19024.539} C_VEL
LIN {X 0,Y 410.909,Z 620.31,A -85,B 0,C 180,E1 19023.61,E2 19023.61} C_VEL
LIN {X 0,Y 408.749,Z 640.92,A -85,B 0,C 180,E1 19022.39,E2 19022.39} C_VEL
LIN {X 0,Y 406.395,Z 660.376,A -85,B 0,C 180,E1 19020.942,E2 19020.942} C_VEL
LIN {X 0,Y 403.973,Z 678.786,A -85,B 0,C 180,E1 19019.261,E2 19019.261} C_VEL
LIN {X 0,Y 401.555,Z 696.152,A -85,B 0,C 180,E1 19017.346,E2 19017.346} C_VEL
LIN {X 0,Y 399.377,Z 711.376,A -85,B 0,C 180,E1 19015.341,E2 19015.341} C_VEL
LIN {X 0,Y 397.371,Z 725.681,A -85,B 0,C 180,E1 19013.11,E2 19013.11} C_VEL
LIN {X 0,Y 395.647,Z 738.602,A -85,B 0,C 180,E1 19010.718,E2 19010.718} C_VEL
LIN {X 0,Y 394.254,Z 750.119,A -85,B 0,C 180,E1 19008.174,E2 19008.174} C_VEL
LIN {X 0,Y 393.264,Z 759.694,A -85,B 0,C 180,E1 19005.633,E2 19005.633} C_VEL
LIN {X 0,Y 392.539,Z 768.289,A -85,B 0,C 180,E1 19002.801,E2 19002.801} C_VEL
LIN {X 0,Y 392.165,Z 774.955,A -85,B 0,C 180,E1 18999.982,E2 18999.982} C_VEL
LIN {X 0,Y 392.007,Z 779.883,A -85,B 0,C 180,E1 18997.169,E2 18997.169} C_VEL
LIN {X 0,Y 391.988,Z 783.143,A -85,B 0,C 180,E1 18994.387,E2 18994.387} C_VEL
LIN {X 0,Y 391.999,Z 784.826,A -85,B 0,C 180,E1 18991.606,E2 18991.606} C_VEL
LIN {X 0,Y 392.011,Z 784.855,A -85,B 0,C 180,E1 18988.928,E2 18988.928} C_VEL
LIN {X 0,Y 392.001,Z 783.287,A -85,B 0,C 180,E1 18986.05,E2 18986.05} C_VEL
LIN {X 0,Y 392.02,Z 780.159,A -85,B 0,C 180,E1 18983.261,E2 18983.261} C_VEL
LIN {X 0,Y 392.132,Z 775.337,A -85,B 0,C 180,E1 18980.458,E2 18980.458} C_VEL
LIN {X 0,Y 392.433,Z 769.064,A -85,B 0,C 180,E1 18977.79,E2 18977.79} C_VEL
LIN {X 0,Y 393.049,Z 760.59,A -85,B 0,C 180,E1 18974.96,E2 18974.96} C_VEL
LIN {X 0,Y 393.982,Z 750.577,A -85,B 0,C 180,E1 18972.268,E2 18972.268} C_VEL
LIN {X 0,Y 395.262,Z 739.097,A -85,B 0,C 180,E1 18969.722,E2 18969.722} C_VEL
LIN {X 0,Y 396.852,Z 726.19,A -85,B 0,C 180,E1 18967.325,E2 18967.325} C_VEL
LIN {X 0,Y 398.795,Z 711.301,A -85,B 0,C 180,E1 18965.008,E2 18965.008} C_VEL
LIN {X 0,Y 401.008,Z 694.704,A -85,B 0,C 180,E1 18962.851,E2 18962.851} C_VEL
LIN {X 0,Y 403.385,Z 676.518,A -85,B 0,C 180,E1 18960.884,E2 18960.884} C_VEL
LIN {X 0,Y 405.775,Z 657.251,A -85,B 0,C 180,E1 18959.166,E2 18959.166} C_VEL
LIN {X 0,Y 408.122,Z 636.959,A -85,B 0,C 180,E1 18957.694,E2 18957.694} C_VEL
LIN {X 0,Y 410.254,Z 616.233,A -85,B 0,C 180,E1 18956.493,E2 18956.493} C_VEL
LIN {X 0,Y 412.2,Z 594.587,A -85,B 0,C 180,E1 18955.531,E2 18955.531} C_VEL
LIN {X 0,Y 413.812,Z 572.25,A -85,B 0,C 180,E1 18954.816,E2 18954.816} C_VEL
LIN {X 0,Y 418.128,Z 493.872,A -85,B 0,C 180,E1 18952.91,E2 18952.91} C_VEL
LIN {X 0,Y 423.367,Z 428.006,A -85,B 0,C 180,E1 18951.135,E2 18951.135} C_VEL
LIN {X 0,Y 430.317,Z 363.895,A -85,B 0,C 180,E1 18949.27,E2 18949.27} C_VEL
LIN {X 0,Y 431.806,Z 351.842,A -85,B 0,C 180,E1 18948.902,E2 18948.902} C_VEL
LIN {X 0,Y 429.203,Z 345.73,A -85,B 0,C 180,E1 18947.75,E2 18947.75} C_VEL
LIN {X 0,Y 426.845,Z 341.145,A -85,B 0,C 180,E1 18946.433,E2 18946.433} C_VEL
LIN {X 0,Y 424.814,Z 337.789,A -85,B 0,C 180,E1 18944.507,E2 18944.507} C_VEL
LIN {X 0,Y 424.298,Z 337.772,A -85,B 0,C 180,E1 18943.266,E2 18943.266} C_VEL
LIN {X 0,Y 424.813,Z 340.3,A -85,B 0,C 180,E1 18941.338,E2 18941.338} C_VEL
LIN {X 0,Y 426.33,Z 344.624,A -85,B 0,C 180,E1 18939.811,E2 18939.811} C_VEL
LIN {X 0,Y 428.359,Z 350.001,A -85,B 0,C 180,E1 18938.506,E2 18938.506} C_VEL
LIN {X 0,Y 429.496,Z 353.537,A -85,B 0,C 180,E1 18937.878,E2 18937.878} C_VEL
LIN {X 0,Y 429.664,Z 372.072,A -85,B 0,C 180,E1 18936.583,E2 18936.583} C_VEL
LIN {X 0,Y 429.502,Z 378.771,A -85,B 0,C 180,E1 18936.218,E2 18936.218} C_VEL
LIN {X 0,Y 420.852,Z 453.997,A -85,B 0,C 180,E1 18933.964,E2 18933.964} C_VEL
LIN {X 0,Y 414.952,Z 523.412,A -85,B 0,C 180,E1 18931.984,E2 18931.984} C_VEL
LIN {X 0,Y 411.775,Z 569.755,A -85,B 0,C 180,E1 18930.691,E2 18930.691} C_VEL
LIN {X 0,Y 410.048,Z 589.973,A -85,B 0,C 180,E1 18929.87,E2 18929.87} C_VEL
LIN {X 0,Y 408.054,Z 609.913,A -85,B 0,C 180,E1 18928.792,E2 18928.792} C_VEL
LIN {X 0,Y 405.951,Z 628.582,A -85,B 0,C 180,E1 18927.504,E2 18927.504} C_VEL
LIN {X 0,Y 403.72,Z 646.478,A -85,B 0,C 180,E1 18925.97,E2 18925.97} C_VEL
LIN {X 0,Y 401.544,Z 662.795,A -85,B 0,C 180,E1 18924.258,E2 18924.258} C_VEL
LIN {X 0,Y 399.466,Z 677.763,A -85,B 0,C 180,E1 18922.361,E2 18922.361} C_VEL
LIN {X 0,Y 397.58,Z 691.237,A -85,B 0,C 180,E1 18920.307,E2 18920.307} C_VEL
LIN {X 0,Y 395.933,Z 703.264,A -85,B 0,C 180,E1 18918.096,E2 18918.096} C_VEL
LIN {X 0,Y 394.567,Z 713.847,A -85,B 0,C 180,E1 18915.732,E2 18915.732} C_VEL
LIN {X 0,Y 393.512,Z 722.946,A -85,B 0,C 180,E1 18913.219,E2 18913.219} C_VEL
LIN {X 0,Y 392.803,Z 730.143,A -85,B 0,C 180,E1 18910.708,E2 18910.708} C_VEL
LIN {X 0,Y 392.356,Z 735.897,A -85,B 0,C 180,E1 18908.057,E2 18908.057} C_VEL
LIN {X 0,Y 392.136,Z 739.907,A -85,B 0,C 180,E1 18905.413,E2 18905.413} C_VEL
LIN {X 0,Y 392.039,Z 742.339,A -85,B 0,C 180,E1 18902.631,E2 18902.631} C_VEL
LIN {X 0,Y 392.022,Z 743.022,A -85,B 0,C 180,E1 18899.999,E2 18899.999} C_VEL
LIN {X 0,Y 392.027,Z 742.021,A -85,B 0,C 180,E1 18897.222,E2 18897.222} C_VEL
LIN {X 0,Y 392.1,Z 739.253,A -85,B 0,C 180,E1 18894.439,E2 18894.439} C_VEL
LIN {X 0,Y 392.314,Z 734.637,A -85,B 0,C 180,E1 18891.646,E2 18891.646} C_VEL
LIN {X 0,Y 392.742,Z 728.456,A -85,B 0,C 180,E1 18888.992,E2 18888.992} C_VEL
LIN {X 0,Y 393.485,Z 720.325,A -85,B 0,C 180,E1 18886.33,E2 18886.33} C_VEL
LIN {X 0,Y 394.55,Z 710.631,A -85,B 0,C 180,E1 18883.813,E2 18883.813} C_VEL
LIN {X 0,Y 395.927,Z 699.422,A -85,B 0,C 180,E1 18881.446,E2 18881.446} C_VEL
LIN {X 0,Y 397.59,Z 686.704,A -85,B 0,C 180,E1 18879.231,E2 18879.231} C_VEL
LIN {X 0,Y 399.492,Z 672.419,A -85,B 0,C 180,E1 18877.173,E2 18877.173} C_VEL
LIN {X 0,Y 401.465,Z 657.392,A -85,B 0,C 180,E1 18875.375,E2 18875.375} C_VEL
LIN {X 0,Y 403.508,Z 640.935,A -85,B 0,C 180,E1 18873.748,E2 18873.748} C_VEL
LIN {X 0,Y 405.56,Z 622.985,A -85,B 0,C 180,E1 18872.307,E2 18872.307} C_VEL
LIN {X 0,Y 407.476,Z 603.872,A -85,B 0,C 180,E1 18871.092,E2 18871.092} C_VEL
LIN {X 0,Y 409.102,Z 584.185,A -85,B 0,C 180,E1 18870.138,E2 18870.138} C_VEL
LIN {X 0,Y 410.384,Z 564.626,A -85,B 0,C 180,E1 18869.463,E2 18869.463} C_VEL
LIN {X 0,Y 411.678,Z 531.02,A -85,B 0,C 180,E1 18868.72,E2 18868.72} C_VEL
LIN {X 0,Y 417.674,Z 373.67,A -85,B 0,C 180,E1 18865.392,E2 18865.392} C_VEL
LIN {X 0,Y 412.809,Z 339.814,A -85,B 0,C 180,E1 18864.051,E2 18864.051} C_VEL
LIN {X 0,Y 412.541,Z 337.856,A -85,B 0,C 180,E1 18863.813,E2 18863.813} C_VEL
LIN {X 0,Y 406.059,Z 319.468,A -85,B 0,C 180,E1 18860.976,E2 18860.976} C_VEL
LIN {X 0,Y 398.94,Z 301.069,A -85,B 0,C 180,E1 18857.892,E2 18857.892} C_VEL
LIN {X 0,Y 393.582,Z 287.659,A -85,B 0,C 180,E1 18855.444,E2 18855.444} C_VEL
LIN {X 0,Y 393.563,Z 287.462,A -85,B 0,C 180,E1 18851.456,E2 18851.456} C_VEL
LIN {X 0,Y 393.56,Z 287.462,A -85,B 0,C 180,E1 18847.565,E2 18847.565} C_VEL
LIN {X 0,Y 393.564,Z 287.463,A -85,B 0,C 180,E1 18843.56,E2 18843.56} C_VEL
LIN {X 0,Y 393.559,Z 287.441,A -85,B 0,C 180,E1 18839.531,E2 18839.531} C_VEL
LIN {X 0,Y 393.552,Z 287.446,A -85,B 0,C 180,E1 18835.588,E2 18835.588} C_VEL
LIN {X 0,Y 393.548,Z 287.449,A -85,B 0,C 180,E1 18831.618,E2 18831.618} C_VEL
LIN {X 0,Y 393.536,Z 287.554,A -85,B 0,C 180,E1 18828.826,E2 18828.826} C_VEL
LIN {X 0,Y 393.987,Z 289.28,A -85,B 0,C 180,E1 18828.497,E2 18828.497} C_VEL
LIN {X 0,Y 401.135,Z 306.789,A -85,B 0,C 180,E1 18825.989,E2 18825.989} C_VEL
LIN {X 0,Y 407.641,Z 325.401,A -85,B 0,C 180,E1 18823.533,E2 18823.533} C_VEL
LIN {X 0,Y 407.824,Z 328.938,A -85,B 0,C 180,E1 18823.172,E2 18823.172} C_VEL
LIN {X 0,Y 406.05,Z 334.761,A -85,B 0,C 180,E1 18822.766,E2 18822.766} C_VEL
LIN {X 0,Y 402.635,Z 343.48,A -85,B 0,C 180,E1 18822.222,E2 18822.222} C_VEL
LIN {X 0,Y 402.207,Z 346.122,A -85,B 0,C 180,E1 18822.001,E2 18822.001} C_VEL
LIN {X 0,Y 399.838,Z 387.755,A -85,B 0,C 180,E1 18818.124,E2 18818.124} C_VEL
LIN {X 0,Y 397.374,Z 430.242,A -85,B 0,C 180,E1 18814.186,E2 18814.186} C_VEL
LIN {X 0,Y 394.991,Z 472.14,A -85,B 0,C 180,E1 18810.292,E2 18810.292} C_VEL
LIN {X 0,Y 394.7,Z 479.497,A -85,B 0,C 180,E1 18809.643,E2 18809.643} C_VEL
LIN {X 0,Y 396.483,Z 496.869,A -85,B 0,C 180,E1 18809.182,E2 18809.182} C_VEL
LIN {X 0,Y 394.065,Z 622.743,A -85,B 0,C 180,E1 18806.824,E2 18806.824} C_VEL
LIN {X 0,Y 393.45,Z 638.836,A -85,B 0,C 180,E1 18806.254,E2 18806.254} C_VEL
LIN {X 0,Y 392.507,Z 654.948,A -85,B 0,C 180,E1 18805.399,E2 18805.399} C_VEL
LIN {X 0,Y 391.39,Z 669.303,A -85,B 0,C 180,E1 18804.357,E2 18804.357} C_VEL
LIN {X 0,Y 390.069,Z 683.635,A -85,B 0,C 180,E1 18803.008,E2 18803.008} C_VEL
LIN {X 0,Y 388.772,Z 696.257,A -85,B 0,C 180,E1 18801.498,E2 18801.498} C_VEL
LIN {X 0,Y 387.5,Z 707.934,A -85,B 0,C 180,E1 18799.746,E2 18799.746} C_VEL
LIN {X 0,Y 386.423,Z 717.792,A -85,B 0,C 180,E1 18797.904,E2 18797.904} C_VEL
LIN {X 0,Y 385.467,Z 726.899,A -85,B 0,C 180,E1 18795.736,E2 18795.736} C_VEL
LIN {X 0,Y 384.8,Z 734.119,A -85,B 0,C 180,E1 18793.5,E2 18793.5} C_VEL
LIN {X 0,Y 384.362,Z 739.874,A -85,B 0,C 180,E1 18791.026,E2 18791.026} C_VEL
LIN {X 0,Y 384.158,Z 743.496,A -85,B 0,C 180,E1 18788.632,E2 18788.632} C_VEL
LIN {X 0,Y 384.083,Z 745.361,A -85,B 0,C 180,E1 18786.205,E2 18786.205} C_VEL
LIN {X 0,Y 384.087,Z 745.527,A -85,B 0,C 180,E1 18783.902,E2 18783.902} C_VEL
LIN {X 0,Y 384.166,Z 743.839,A -85,B 0,C 180,E1 18781.389,E2 18781.389} C_VEL
LIN {X 0,Y 384.38,Z 740.5,A -85,B 0,C 180,E1 18779.002,E2 18779.002} C_VEL
LIN {X 0,Y 384.766,Z 735.571,A -85,B 0,C 180,E1 18776.751,E2 18776.751} C_VEL
LIN {X 0,Y 385.43,Z 728.74,A -85,B 0,C 180,E1 18774.476,E2 18774.476} C_VEL
LIN {X 0,Y 386.342,Z 720.344,A -85,B 0,C 180,E1 18772.357,E2 18772.357} C_VEL
LIN {X 0,Y 387.506,Z 710.223,A -85,B 0,C 180,E1 18770.351,E2 18770.351} C_VEL
LIN {X 0,Y 388.761,Z 699.273,A -85,B 0,C 180,E1 18768.628,E2 18768.628} C_VEL
LIN {X 0,Y 390.138,Z 686.536,A -85,B 0,C 180,E1 18767.025,E2 18767.025} C_VEL
LIN {X 0,Y 391.426,Z 673.431,A -85,B 0,C 180,E1 18765.716,E2 18765.716} C_VEL
LIN {X 0,Y 392.715,Z 658.035,A -85,B 0,C 180,E1 18764.533,E2 18764.533} C_VEL
LIN {X 0,Y 393.695,Z 642.674,A -85,B 0,C 180,E1 18763.66,E2 18763.66} C_VEL
LIN {X 0,Y 394.411,Z 625.713,A -85,B 0,C 180,E1 18763.007,E2 18763.007} C_VEL
LIN {X 0,Y 394.914,Z 601.292,A -85,B 0,C 180,E1 18762.492,E2 18762.492} C_VEL
LIN {X 0,Y 396.897,Z 494.063,A -85,B 0,C 180,E1 18760.484,E2 18760.484} C_VEL
LIN {X 0,Y 395.229,Z 479.296,A -85,B 0,C 180,E1 18760.032,E2 18760.032} C_VEL
LIN {X 0,Y 397.566,Z 436.543,A -85,B 0,C 180,E1 18756.105,E2 18756.105} C_VEL
LIN {X 0,Y 399.816,Z 396.458,A -85,B 0,C 180,E1 18752.441,E2 18752.441} C_VEL
LIN {X 0,Y 401.861,Z 357.064,A -85,B 0,C 180,E1 18748.862,E2 18748.862} C_VEL
LIN {X 0,Y 402.887,Z 334.115,A -85,B 0,C 180,E1 18746.772,E2 18746.772} C_VEL
LIN {X 0,Y 397.283,Z 316.981,A -85,B 0,C 180,E1 18744.536,E2 18744.536} C_VEL
LIN {X 0,Y 390.583,Z 299.994,A -85,B 0,C 180,E1 18742.106,E2 18742.106} C_VEL
LIN {X 0,Y 386.577,Z 291.412,A -85,B 0,C 180,E1 18740.754,E2 18740.754} C_VEL
LIN {X 0,Y 385.632,Z 288.744,A -85,B 0,C 180,E1 18740.291,E2 18740.291} C_VEL
LIN {X 0,Y 385.591,Z 288.444,A -85,B 0,C 180,E1 18738.287,E2 18738.287} C_VEL
LIN {X 0,Y 385.59,Z 288.452,A -85,B 0,C 180,E1 18734.262,E2 18734.262} C_VEL
LIN {X 0,Y 385.591,Z 288.453,A -85,B 0,C 180,E1 18730.307,E2 18730.307} C_VEL
LIN {X 0,Y 385.59,Z 288.45,A -85,B 0,C 180,E1 18726.253,E2 18726.253} C_VEL
LIN {X 0,Y 385.59,Z 288.455,A -85,B 0,C 180,E1 18722.23,E2 18722.23} C_VEL
LIN {X 0,Y 385.591,Z 288.45,A -85,B 0,C 180,E1 18718.217,E2 18718.217} C_VEL
LIN {X 0,Y 385.592,Z 288.454,A -85,B 0,C 180,E1 18714.196,E2 18714.196} C_VEL
LIN {X 0,Y 385.593,Z 288.446,A -85,B 0,C 180,E1 18710.146,E2 18710.146} C_VEL
LIN {X 0,Y 385.594,Z 288.452,A -85,B 0,C 180,E1 18706.046,E2 18706.046} C_VEL
LIN {X 0,Y 385.596,Z 288.453,A -85,B 0,C 180,E1 18702.027,E2 18702.027} C_VEL
LIN {X 0,Y 385.593,Z 288.447,A -85,B 0,C 180,E1 18698.075,E2 18698.075} C_VEL
LIN {X 0,Y 385.597,Z 288.453,A -85,B 0,C 180,E1 18694.01,E2 18694.01} C_VEL
LIN {X 0,Y 385.6,Z 288.449,A -85,B 0,C 180,E1 18689.971,E2 18689.971} C_VEL
LIN {X 0,Y 385.6,Z 288.45,A -85,B 0,C 180,E1 18685.939,E2 18685.939} C_VEL
LIN {X 0,Y 385.601,Z 288.45,A -85,B 0,C 180,E1 18681.894,E2 18681.894} C_VEL
LIN {X 0,Y 385.659,Z 288.721,A -85,B 0,C 180,E1 18678.472,E2 18678.472} C_VEL
LIN {X 0,Y 388.596,Z 295.735,A -85,B 0,C 180,E1 18677.161,E2 18677.161} C_VEL
LIN {X 0,Y 397.618,Z 316.933,A -85,B 0,C 180,E1 18673.597,E2 18673.597} C_VEL
LIN {X 0,Y 398.948,Z 319.876,A -85,B 0,C 180,E1 18673.198,E2 18673.198} C_VEL
LIN {X 0,Y 414.538,Z 347.5,A -85,B 0,C 180,E1 18670.821,E2 18670.821} C_VEL
LIN {X 0,Y 416.358,Z 351.397,A -85,B 0,C 180,E1 18670.539,E2 18670.539} C_VEL
LIN {X 0,Y 408.437,Z 546.701,A -85,B 0,C 180,E1 18666.458,E2 18666.458} C_VEL
LIN {X 0,Y 407.015,Z 580.064,A -85,B 0,C 180,E1 18665.71,E2 18665.71} C_VEL
LIN {X 0,Y 405.492,Z 601.047,A -85,B 0,C 180,E1 18664.994,E2 18664.994} C_VEL
LIN {X 0,Y 403.586,Z 621.322,A -85,B 0,C 180,E1 18664.047,E2 18664.047} C_VEL
LIN {X 0,Y 401.48,Z 640.647,A -85,B 0,C 180,E1 18662.88,E2 18662.88} C_VEL
LIN {X 0,Y 399.03,Z 660.122,A -85,B 0,C 180,E1 18661.41,E2 18661.41} C_VEL
LIN {X 0,Y 396.51,Z 678.559,A -85,B 0,C 180,E1 18659.701,E2 18659.701} C_VEL
LIN {X 0,Y 394.072,Z 695.297,A -85,B 0,C 180,E1 18657.828,E2 18657.828} C_VEL
LIN {X 0,Y 391.716,Z 711.133,A -85,B 0,C 180,E1 18655.715,E2 18655.715} C_VEL
LIN {X 0,Y 389.616,Z 725.484,A -85,B 0,C 180,E1 18653.437,E2 18653.437} C_VEL
LIN {X 0,Y 387.808,Z 738.415,A -85,B 0,C 180,E1 18650.998,E2 18650.998} C_VEL
LIN {X 0,Y 386.351,Z 749.923,A -85,B 0,C 180,E1 18648.403,E2 18648.403} C_VEL
LIN {X 0,Y 385.269,Z 759.915,A -85,B 0,C 180,E1 18645.673,E2 18645.673} C_VEL
LIN {X 0,Y 384.53,Z 768.479,A -85,B 0,C 180,E1 18642.767,E2 18642.767} C_VEL
LIN {X 0,Y 384.157,Z 775.03,A -85,B 0,C 180,E1 18639.89,E2 18639.89} C_VEL
LIN {X 0,Y 384.012,Z 779.583,A -85,B 0,C 180,E1 18637.178,E2 18637.178} C_VEL
LIN {X 0,Y 383.999,Z 782.86,A -85,B 0,C 180,E1 18634.249,E2 18634.249} C_VEL
LIN {X 0,Y 384.011,Z 784.423,A -85,B 0,C 180,E1 18631.49,E2 18631.49} C_VEL
LIN {X 0,Y 384.02,Z 784.396,A -85,B 0,C 180,E1 18628.805,E2 18628.805} C_VEL
LIN {X 0,Y 384.009,Z 782.846,A -85,B 0,C 180,E1 18625.967,E2 18625.967} C_VEL
LIN {X 0,Y 384.024,Z 779.703,A -85,B 0,C 180,E1 18623.12,E2 18623.12} C_VEL
LIN {X 0,Y 384.151,Z 774.855,A -85,B 0,C 180,E1 18620.258,E2 18620.258} C_VEL
LIN {X 0,Y 384.471,Z 768.554,A -85,B 0,C 180,E1 18617.533,E2 18617.533} C_VEL
LIN {X 0,Y 385.142,Z 760.046,A -85,B 0,C 180,E1 18614.643,E2 18614.643} C_VEL
LIN {X 0,Y 386.17,Z 749.788,A -85,B 0,C 180,E1 18611.845,E2 18611.845} C_VEL
LIN {X 0,Y 387.524,Z 738.476,A -85,B 0,C 180,E1 18609.298,E2 18609.298} C_VEL
LIN {X 0,Y 389.231,Z 725.53,A -85,B 0,C 180,E1 18606.856,E2 18606.856} C_VEL
LIN {X 0,Y 391.309,Z 710.607,A -85,B 0,C 180,E1 18604.496,E2 18604.496} C_VEL
LIN {X 0,Y 393.671,Z 693.985,A -85,B 0,C 180,E1 18602.302,E2 18602.302} C_VEL
LIN {X 0,Y 396.149,Z 676.253,A -85,B 0,C 180,E1 18600.349,E2 18600.349} C_VEL
LIN {X 0,Y 398.765,Z 656.587,A -85,B 0,C 180,E1 18598.563,E2 18598.563} C_VEL
LIN {X 0,Y 401.223,Z 636.704,A -85,B 0,C 180,E1 18597.093,E2 18597.093} C_VEL
LIN {X 0,Y 403.581,Z 615.51,A -85,B 0,C 180,E1 18595.84,E2 18595.84} C_VEL
LIN {X 0,Y 405.687,Z 593.804,A -85,B 0,C 180,E1 18594.854,E2 18594.854} C_VEL
LIN {X 0,Y 407.476,Z 571.241,A -85,B 0,C 180,E1 18594.115,E2 18594.115} C_VEL
LIN {X 0,Y 412.132,Z 497.627,A -85,B 0,C 180,E1 18592.233,E2 18592.233} C_VEL
LIN {X 0,Y 417.762,Z 434.94,A -85,B 0,C 180,E1 18590.468,E2 18590.468} C_VEL
LIN {X 0,Y 425.447,Z 371.518,A -85,B 0,C 180,E1 18588.554,E2 18588.554} C_VEL
LIN {X 0,Y 427.584,Z 355.86,A -85,B 0,C 180,E1 18588.039,E2 18588.039} C_VEL
LIN {X 0,Y 425.739,Z 351.406,A -85,B 0,C 180,E1 18587.051,E2 18587.051} C_VEL
LIN {X 0,Y 424.157,Z 348.165,A -85,B 0,C 180,E1 18585.969,E2 18585.969} C_VEL
LIN {X 0,Y 422.802,Z 345.516,A -85,B 0,C 180,E1 18584.423,E2 18584.423} C_VEL
LIN {X 0,Y 422.342,Z 345.513,A -85,B 0,C 180,E1 18583.357,E2 18583.357} C_VEL
LIN {X 0,Y 422.646,Z 347.936,A -85,B 0,C 180,E1 18581.528,E2 18581.528} C_VEL
LIN {X 0,Y 423.852,Z 352.079,A -85,B 0,C 180,E1 18580.059,E2 18580.059} C_VEL
LIN {X 0,Y 425.435,Z 357.078,A -85,B 0,C 180,E1 18578.866,E2 18578.866} C_VEL
LIN {X 0,Y 425.847,Z 358.986,A -85,B 0,C 180,E1 18578.557,E2 18578.557} C_VEL
